	10://Clear old Data on GVL 	
		Lynus_Standards.GVL_Energy.stDataElectricHeatingElements[diNrOfEMS_IN_CP,diNrOfEHE_OUT].bEnabled := FALSE;
			Lynus_Standards.GVL_Energy.stDataElectricHeatingElements[diNrOfEMS_IN_CP,diNrOfEHE_OUT].bIsStepSwitched := FALSE;
				Lynus_Standards.GVL_Energy.stDataElectricHeatingElements[diNrOfEMS_IN_CP,diNrOfEHE_OUT].bIsControllable := FALSE;
					Lynus_Standards.GVL_Energy.stDataElectricHeatingElements[diNrOfEMS_IN_CP,diNrOfEHE_OUT].byPriority := 0;
						Lynus_Standards.GVL_Energy.stDataElectricHeatingElements[diNrOfEMS_IN_CP,diNrOfEHE_OUT].byErrorWarning := 0;
							Lynus_Standards.GVL_Energy.stDataElectricHeatingElements[diNrOfEMS_IN_CP,diNrOfEHE_OUT].byNumberOfSteps := 0;
								Lynus_Standards.GVL_Energy.stDataElectricHeatingElements[diNrOfEMS_IN_CP,diNrOfEHE_OUT].lrPower := 0;
									Lynus_Standards.GVL_Energy.stDataElectricHeatingElements[diNrOfEMS_IN_CP,diNrOfEHE_OUT].lrPowerConsumption := 0;
										Lynus_Standards.GVL_Energy.stDataElectricHeatingElements[diNrOfEMS_IN_CP,diNrOfEHE_OUT].lrPowerProduction := 0;
											FOR byLPGVLSetMaxPower := 1 TO 10 BY 1 DO
												Lynus_Standards.GVL_Energy.stDataElectricHeatingElements[diNrOfEMS_IN_CP,diNrOfEHE_OUT].arrMaxPower[byLPGVLSetMaxPower] := 0;
											END_FOR 
												
		diNrOfEMS_IN_CP := diNrOfEMS_IN;
			//Back to the init step
			iStateGVLData := 0;

END_CASE 	 

IF diNrOfEHE_OUT > 0 AND fbNumberDevice.bNumberIsCalculatet AND diNrOfEMS_IN > 0 THEN
	Lynus_Standards.GVL_Energy.stDataElectricHeatingElements[diNrOfEMS_IN,diNrOfEHE_OUT].bEnabled := fbEHE.stDataEHEOut.bEnabled;
		Lynus_Standards.GVL_Energy.stDataElectricHeatingElements[diNrOfEMS_IN,diNrOfEHE_OUT].bIsStepSwitched := fbEHE.stDataEHEOut.bIsStepSwitched;
			Lynus_Standards.GVL_Energy.stDataElectricHeatingElements[diNrOfEMS_IN,diNrOfEHE_OUT].bIsControllable := TRUE;
				Lynus_Standards.GVL_Energy.stDataElectricHeatingElements[diNrOfEMS_IN,diNrOfEHE_OUT].byPriority := fbEHE.stDataEHEOut.byPriority;
					Lynus_Standards.GVL_Energy.stDataElectricHeatingElements[diNrOfEMS_IN,diNrOfEHE_OUT].byErrorWarning := fbEHE.stDataEHEOut.byErrorWarning;
						Lynus_Standards.GVL_Energy.stDataElectricHeatingElements[diNrOfEMS_IN,diNrOfEHE_OUT].byNumberOfSteps := fbEHE.stDataEHEOut.byNumberOfSteps;
							Lynus_Standards.GVL_Energy.stDataElectricHeatingElements[diNrOfEMS_IN,diNrOfEHE_OUT].lrPower := fbEHE.stDataEHEOut.lrPower;
								Lynus_Standards.GVL_Energy.stDataElectricHeatingElements[diNrOfEMS_IN,diNrOfEHE_OUT].lrPowerConsumption := fbEHE.stDataEHEOut.lrPowerConsumption;
									Lynus_Standards.GVL_Energy.stDataElectricHeatingElements[diNrOfEMS_IN,diNrOfEHE_OUT].lrPowerProduction := fbEHE.stDataEHEOut.lrPowerProduction;
										Lynus_Standards.GVL_Energy.stDataElectricHeatingElements[diNrOfEMS_IN,diNrOfEHE_OUT].arrMaxPower := fbEHE.stDataEHEOut.arrMaxPower;
END_IF			
		
(*----------------------------------------------------------Save persistent data----------------------------------------------------------------*)

arrPD[1](lrValue:= BOOL_TO_LREAL(bEnable), bEventBasedActive=> );
arrPD[2](lrValue:= BOOL_TO_LREAL(bPowerDataInvers), bEventBasedActive=> );
arrPD[3](lrValue:= DINT_TO_LREAL(diNrOfEMS_IN), bEventBasedActive=> );
arrPD[4](lrValue:= DINT_TO_LREAL(diNrOfEM_IN_EHE), bEventBasedActive=> );
arrPD[5](lrValue:= DINT_TO_LREAL(diNrOfTempS_IN), bEventBasedActive=> );
arrPD[6](lrValue:= REAL_TO_LREAL(stSetupEHE.rMaxPower1), bEventBasedActive=> );
arrPD[7](lrValue:= REAL_TO_LREAL(stSetupEHE.rMaxPower2), bEventBasedActive=> );
arrPD[8](lrValue:= REAL_TO_LREAL(stSetupEHE.rMaxPower3), bEventBasedActive=> );
arrPD[9](lrValue:= REAL_TO_LREAL(stSetupEHE.rMaxPower4), bEventBasedActive=> );
arrPD[10](lrValue:= REAL_TO_LREAL(stSetupEHE.rMaxPower5), bEventBasedActive=> );
arrPD[11](lrValue:= REAL_TO_LREAL(stSetupEHE.rMaxPower6), bEventBasedActive=> );
arrPD[12](lrValue:= REAL_TO_LREAL(stSetupEHE.rMaxPower7), bEventBasedActive=> );
arrPD[13](lrValue:= REAL_TO_LREAL(stSetupEHE.rMaxPower8), bEventBasedActive=> );
arrPD[14](lrValue:= REAL_TO_LREAL(stSetupEHE.rMaxPower9), bEventBasedActive=> );
arrPD[15](lrValue:= REAL_TO_LREAL(stSetupEHE.rMaxPower10), bEventBasedActive=> );
arrPD[16](lrValue:= BOOL_TO_LREAL(stSetupEHE.bDisableLegionellaPr), bEventBasedActive=> );
arrPD[17](lrValue:= BOOL_TO_LREAL(stSetupEHE.bManualyOn), bEventBasedActive=> );
arrPD[18](lrValue:= BOOL_TO_LREAL(stSetupEHE.bOnEmergPowerOff), bEventBasedActive=> );
arrPD[19](lrValue:= BOOL_TO_LREAL(stSetupEHE.bTimeEnabled), bEventBasedActive=> );
arrPD[20](lrValue:= BYTE_TO_LREAL(stSetupEHE.byDisableSOC), bEventBasedActive=> );
arrPD[21](lrValue:= BYTE_TO_LREAL(stSetupEHE.byEnableSOC), bEventBasedActive=> );
arrPD[22](lrValue:= BYTE_TO_LREAL(stSetupEHE.byHourOff), bEventBasedActive=> );
arrPD[23](lrValue:= BYTE_TO_LREAL(stSetupEHE.byHourOn), bEventBasedActive=> );
arrPD[24](lrValue:= BYTE_TO_LREAL(stSetupEHE.byManualyTargetPower), bEventBasedActive=> );
arrPD[25](lrValue:= BYTE_TO_LREAL(stSetupEHE.byMinutesOff), bEventBasedActive=> );
arrPD[26](lrValue:= BYTE_TO_LREAL(stSetupEHE.byMinutesOn), bEventBasedActive=> );
arrPD[27](lrValue:= BYTE_TO_LREAL(stSetupEHE.byPriority), bEventBasedActive=> );
arrPD[28](lrValue:= UINT_TO_LREAL(stSetupEHE.uiTargetTempMax), bEventBasedActive=> );
arrPD[29](lrValue:= UINT_TO_LREAL(stSetupEHE.uiTargetTempOff), bEventBasedActive=> );
arrPD[30](lrValue:= UINT_TO_LREAL(stSetupEHE.uiTargetTempOn), bEventBasedActive=> );
arrPD[31](lrValue:= DINT_TO_LREAL(diNrOfEMS_IN_CP), bEventBasedActive=> );
arrPD[32](lrValue:= BOOL_TO_LREAL(bNoLinear), bEventBasedActive=> );
arrPD[33](lrValue:= REAL_TO_LREAL(arrTableOfInterpolationPoints[1]), bEventBasedActive=> );
arrPD[34](lrValue:= REAL_TO_LREAL(arrTableOfInterpolationPoints[2]), bEventBasedActive=> );
arrPD[35](lrValue:= REAL_TO_LREAL(arrTableOfInterpolationPoints[3]), bEventBasedActive=> );
arrPD[36](lrValue:= REAL_TO_LREAL(arrTableOfInterpolationPoints[4]), bEventBasedActive=> );
arrPD[37](lrValue:= REAL_TO_LREAL(arrTableOfInterpolationPoints[5]), bEventBasedActive=> );
arrPD[38](lrValue:= REAL_TO_LREAL(arrTableOfInterpolationPoints[6]), bEventBasedActive=> );
arrPD[39](lrValue:= REAL_TO_LREAL(arrTableOfInterpolationPoints[7]), bEventBasedActive=> );
arrPD[40](lrValue:= REAL_TO_LREAL(arrTableOfInterpolationPoints[8]), bEventBasedActive=> );
arrPD[41](lrValue:= REAL_TO_LREAL(arrTableOfInterpolationPoints[9]), bEventBasedActive=> );
arrPD[42](lrValue:= REAL_TO_LREAL(arrTableOfInterpolationPoints[10]), bEventBasedActive=> );

END_FUNCTION_BLOCK

// ---- FBs/Electric Heating Element/OnOff/FB_EHE_OnOff.TcPOU
FUNCTION_BLOCK FB_EHE_OnOff
VAR_INPUT PERSISTENT
	bEnable									: BOOL;																							//{#lynus.ag#()} //Enable the Fuctionblock and his logic
	bPowerDataInvers						: BOOL;																							//With True its possible to invert all received power data from the electric meter
	diNrOfEMS_IN							: DINT;																							//Number of EMS what control this Device.
	diNrOfEM_IN_EHE							: DINT;																							//Number of the electric meter for incoming power data. (Power Data for this Device)
	diNrOfTempS_IN							: DINT;																							//Number of the Temperature Sensor for incoming temperature data. (Temperature for the Service wather buffer)
	stSetupEHE								: ST_Setup_EHE := (uiTargetTempOn := 35, uiTargetTempOff := 50, uiTargetTempMax := 62);			//{#lynus.ag#()} //Setup electric heating element
END_VAR
VAR_INPUT
END_VAR
VAR_OUTPUT
	stDataEHE								: ST_EHE_Output;																				//{#lynus.ag#()} //Electric heating element output data
	diNrOfEHE_OUT							: DINT;																							//Active Number from the Electric heating element for using on other functions
	rTargetPowerForExtFunc					: REAL;																							//Target Power from 0% to +100% to use on a external Function
END_VAR
VAR
	{attribute 'conditionalshow'}
	fbEHE									: FB_ElectricHeatingElement;																	//Function block for electric heating element
	{attribute 'hide'}
	fbNumberDevice							: FB_NumberOfDevice;																			//Function block to calcualte the number of the Device
	fbDIExternalLock						: FB_XL1XXX_DI;																					//Digital Input from external loock signal
	fbDOOnOffEHE							: FB_XL2XXX_DO;																					//Digital Output to swtich on and off the EHE
	{attribute 'hide'}
	timDissableFunctions					: TON;																							//Timer to dissable the Function after Lynus_Standards.Constants_General.tTimeDissableLynusFunctions Days without connection to the Lynus Cloud
	{attribute 'hide'}
	timResetConnectionOnGVL					: TON;																							//Timer to try reset the connection Flag on the GVL. (When somebody delete the Connection Function and make only a onlinechange)
	{attribute 'hide'}
	timGetTime								: TON;																							//Timer to activate the function tho read out the windows system time
	{attribute 'hide'}
	fbGetSystemTime							: NT_GetTime;																					//Function to read out the windows system time on the local plc
	{attribute 'hide'}
	arrPD									: ARRAY[1..31] OF FB_PersistentData_Number;														//Function to save persistent data 
	{attribute 'hide'}
	byLPTargetPowerTo0						: BYTE;																							//Loop to set the target power from the ems and the max power from the settings for arr[2] to arr[10] to 0 because its only a onOff EHE
	{attribute 'hide'}
	byLPGVLSetMaxPower						: BYTE;																							//Loop to send the max power from the EHE to the GVL
	{attribute 'hide'}
	byWaitInStep							: BYTE;																							//Wait in Step before start to clean data on PLC
	{attribute 'hide'}
	iStateGVLData							: INT;																							//State machine to handle the data on the GVL
	{attribute 'hide'}
	diNumberOfActiveBatterys				: DINT;																							//Number of active batterys
	{attribute 'hide'}
	diNumberOfBatteryInverterInEPO			: DINT;																							//Number of battery inverters that work in Emergency Power operation 
	{attribute 'hide'}
	diCounterForGVL							: DINT;																							//Counter to clean old data on GVL
	{attribute 'hide'}
	diLPForGVL								: DINT;																							//Loop to clean old data on GVL
	{attribute 'hide'}
	dwSumSOC								: DWORD;																						//Sum of the SOC from all batterys
	{attribute 'hide'}
	lrGridPower								: LREAL;																						//Grid power in kW
	{attribute 'hide'}
	lrSizeGridConnection					: LREAL;																						//Size of the complete grid connection
	{attribute 'hide'}
	liLPBatteryData							: LINT;																							//Loop to check some data from batterys
	{attribute 'hide'}
	liLPInEPO								: LINT;																							//Loop to check if 1 or more battery inverters build a island grid
	{attribute 'hide'}
	liLPGridData							: LINT;																							//Loop to check some grid data																				
END_VAR
VAR PERSISTENT
	{attribute 'conditionalshow'}
	diNrOfEMS_IN_CP							: DINT;																							//Number of EMS what control this Device to compare with the original
END_VAR

//Creator : Kai Ebensperger
//Company : Lynus AG
//Date : 19.05.2021
//Version : 1.0.0.0

//With this function block its possible to switch on and off a electric heating element
//The output signal to switch on and off is a digital output signal
//With this function block its not possible to control the EHE with a target power value because we didn't have a active communication to the EHE
//With the Nr from the Electric Meter its possible to send the data fromt the electric meter directly to the EHE function to display it

//NOTE for diNr.....Designation => 
//_IN = Here Data come in from other Functions or go out to other functions about the GVL
//_OUT = Here Data go out to other functions about the GVL

(*------------------------------------------------------------Limits----------------------------------------------------------------------------------*)

diNrOfEMS_IN := LIMIT(0,diNrOfEMS_IN,Constants_Energy.diMaxNumberOfEMS);
	diNrOfEM_IN_EHE := LIMIT(0,diNrOfEM_IN_EHE,Constants_Energy.diMaxNumberOfElectricMeters);
		diNrOfTempS_IN := LIMIT(0,diNrOfTempS_IN,Constants_Sensors.diMaxNumberOfTemperatureSensors);
			
(*------------------------------------------------------------------Power Data----------------------------------------------------------------------------*)

IF NOT bPowerDataInvers THEN
	fbEHE.lrCounterEnergyT1_Consumption := Lynus_Standards.GVL_Energy.stDataElectricMeters[diNrOfEM_IN_EHE].lrCounterEnergyT1_Production * 1000;
	fbEHE.lrCounterEnergyT2_Consumption := Lynus_Standards.GVL_Energy.stDataElectricMeters[diNrOfEM_IN_EHE].lrCounterEnergyT2_Production * 1000;
	fbEHE.lrCounterEnergyT1_Production := Lynus_Standards.GVL_Energy.stDataElectricMeters[diNrOfEM_IN_EHE].lrCounterEnergyT1_Consumption * 1000;
	fbEHE.lrCounterEnergyT2_Production := Lynus_Standards.GVL_Energy.stDataElectricMeters[diNrOfEM_IN_EHE].lrCounterEnergyT1_Consumption * 1000;
	fbEHE.lrTotalCounterEnergy_Consumption := Lynus_Standards.GVL_Energy.stDataElectricMeters[diNrOfEM_IN_EHE].lrTotalCounterEnergy_Production * 1000;
	fbEHE.lrTotalCounterEnergy_Production := Lynus_Standards.GVL_Energy.stDataElectricMeters[diNrOfEM_IN_EHE].lrTotalCounterEnergy_Consumption * 1000;
		fbEHE.lrPowerEHE := (Lynus_Standards.GVL_Energy.stDataElectricMeters[diNrOfEM_IN_EHE].lrPower * 1000) * - 1;
ELSE
	fbEHE.lrCounterEnergyT1_Consumption := Lynus_Standards.GVL_Energy.stDataElectricMeters[diNrOfEM_IN_EHE].lrCounterEnergyT1_Consumption * 1000;
	fbEHE.lrCounterEnergyT2_Consumption := Lynus_Standards.GVL_Energy.stDataElectricMeters[diNrOfEM_IN_EHE].lrCounterEnergyT2_Consumption * 1000;
	fbEHE.lrCounterEnergyT1_Production := Lynus_Standards.GVL_Energy.stDataElectricMeters[diNrOfEM_IN_EHE].lrCounterEnergyT1_Production * 1000;
	fbEHE.lrCounterEnergyT2_Production := Lynus_Standards.GVL_Energy.stDataElectricMeters[diNrOfEM_IN_EHE].lrCounterEnergyT2_Production * 1000;
	fbEHE.lrTotalCounterEnergy_Consumption := Lynus_Standards.GVL_Energy.stDataElectricMeters[diNrOfEM_IN_EHE].lrTotalCounterEnergy_Consumption * 1000;
	fbEHE.lrTotalCounterEnergy_Production := Lynus_Standards.GVL_Energy.stDataElectricMeters[diNrOfEM_IN_EHE].lrTotalCounterEnergy_Production * 1000;
		fbEHE.lrPowerEHE := Lynus_Standards.GVL_Energy.stDataElectricMeters[diNrOfEM_IN_EHE].lrPower * 1000;
END_IF

(*-------------------------------------------------------------Calcualte the number of EHE---------------------------------------------------------------*)

fbNumberDevice(
	diActualNumberOfDevices:= Lynus_Standards.GVL_Energy.stNumberOfDevices.diNumberOfEHE, 
	diMaxNumberOfDevices:= Constants_Energy.diMaxNumberOfElectricHeatingElements, 
	udiCounterOnlineChange:= TwinCAT_SystemInfoVarList._AppInfo.OnlineChangeCnt, 
	bNumberIsCalculatet=> , 
	bFPNumberIsCalculatet=> , 
	bOnlineChange=> , 
	diNumberForThisDevice=> diNrOfEHE_OUT, 
	diNumberOfTotalDevices=> );

//Write new Numer on GVL
IF fbNumberDevice.bFPNumberIsCalculatet THEN
	Lynus_Standards.GVL_Energy.stNumberOfDevices.diNumberOfEHE := fbNumberDevice.diNumberOfTotalDevices;	
END_IF 

//Delete old Number on GVL
IF fbNumberDevice.bOnlineChange THEN 
	Lynus_Standards.GVL_Energy.stNumberOfDevices.diNumberOfEHE := diNrOfEHE_OUT;	
		iStateGVLData := 1; 
END_IF

(*-------------------------------------------------------------Get the local windows system time for this plc---------------------------------------------------------------*)
timGetTime(IN:= bEnable AND NOT timGetTime.Q, PT:= T#30S, Q=> , ET=> );

fbGetSystemTime(
	NETID:= , 
	START:= timGetTime.Q AND NOT fbGetSystemTime.BUSY, 
	TMOUT:= , 
	BUSY=> , 
	ERR=> , 
	ERRID=> , 
	TIMESTR=> );	

fbEHE.stSystemTime.wHour := fbGetSystemTime.TIMESTR.wHour;
	fbEHE.stSystemTime.wMinute := fbGetSystemTime.TIMESTR.wMinute;

(*-------------------------------------------------------------Service from Backend is ready and check the connection to backen for dissabel/enable Function---------------------------------------------------------------*)

//Try to reset the variable for connection on the GVL. When all is normal then the Lynus Mqtt connection function set this variable to true in the next cycle
//When we have no connection to the backend then after Lynus_Standards.Constants_General.tTimeDissableLynusFunctions days the Function is dissabled with all of his functionalities
timResetConnectionOnGVL(IN:= NOT timResetConnectionOnGVL.Q, PT:= T#1H, Q=> , ET=> );
	IF timResetConnectionOnGVL.Q THEN Lynus_Standards.GVL_Communicator.bStateConnectionToEnableFunctions := FALSE; END_IF
		IF NOT Lynus_Standards.GVL_Communicator.bStateConnectionToEnableFunctions THEN timDissableFunctions.IN := TRUE; ELSE timDissableFunctions.IN := FALSE; END_IF  
			timDissableFunctions(IN:= , PT:= Lynus_Standards.Constants_General.tTimeDissableLynusFunctions, Q=> , ET=> );
	
(*------------------------------------------------------------------Error----------------------------------------------------------------------------*)	

IF timDissableFunctions.Q THEN fbEHE.bWarning := TRUE; fbEHE.iWarningCode := 0; ELSE fbEHE.bWarning := FALSE; END_IF 
	IF (Lynus_Standards.GVL_Energy.stNumberOfDevices.diNumberOfEHE > Constants_Energy.diMaxNumberOfElectricHeatingElements) OR 
		(Lynus_Standards.GVL_Sensors.stDataTemperatureSensors[diNrOfTempS_IN].bEnabled AND Lynus_Standards.GVL_Sensors.stDataTemperatureSensors[diNrOfTempS_IN].byErrorWarning = 2) OR
			fbGetSystemTime.ERR THEN 
				fbEHE.bError := TRUE; 
	ELSE 
				fbEHE.bError := FALSE; 
	END_IF

IF Lynus_Standards.GVL_Energy.stNumberOfDevices.diNumberOfEHE > Constants_Energy.diMaxNumberOfElectricHeatingElements THEN fbEHE.iErrorCode := 1;
ELSIF fbGetSystemTime.ERR THEN fbEHE.iErrorCode := 3;
ELSIF Lynus_Standards.GVL_Sensors.stDataTemperatureSensors[diNrOfTempS_IN].bEnabled AND Lynus_Standards.GVL_Sensors.stDataTemperatureSensors[diNrOfTempS_IN].byErrorWarning = 2 THEN fbEHE.iErrorCode := 2;
END_IF

(*------------------------------------------------------------------Logic----------------------------------------------------------------------------*)
	
//Calcualte the total SOC if we have more then 1 battery in our system
diNumberOfActiveBatterys := 0;
	dwSumSOC := 0;
		FOR liLPBatteryData := 1 TO Constants_Energy.diMaxNumberOfBatterys BY 1 DO
			IF Lynus_Standards.GVL_Energy.stDataOfBatterys[diNrOfEMS_IN,liLPBatteryData].bEnabled THEN diNumberOfActiveBatterys := diNumberOfActiveBatterys + 1; END_IF
				dwSumSOC := dwSumSOC + Lynus_Standards.GVL_Energy.stDataOfBatterys[diNrOfEMS_IN,liLPBatteryData].dwSOC;
		END_FOR
	
IF diNumberOfActiveBatterys > 0 THEN
	fbEHE.dwBatterySOC := DINT_TO_DWORD(DWORD_TO_DINT(dwSumSOC) / diNumberOfActiveBatterys);
ELSE
	fbEHE.dwBatterySOC := 100;	//When we have no battery in the ems system
END_IF

//Check if one or more Batterysystems or batteryinverter make island mode
diNumberOfBatteryInverterInEPO := 0;
	FOR liLPInEPO := 1 TO Constants_Energy.diMaxNumberOfBatteryInverters BY 1 DO
		IF Lynus_Standards.GVL_Energy.stDataOfBatteryInverters[diNrOfEMS_IN,liLPInEPO].bWorkOnIslandMode THEN fbEHE.bEPOIsActive := TRUE; diNumberOfBatteryInverterInEPO := diNumberOfBatteryInverterInEPO + 1; END_IF
	END_FOR 
		IF diNumberOfBatteryInverterInEPO <= 0 THEN fbEHE.bEPOIsActive := FALSE; END_IF

//Check the max. power of the grid connection and the sum of grid power
lrSizeGridConnection := 0;
	lrGridPower := 0;
		FOR liLPGridData := 1 TO Constants_Energy.diMaxNumberOfGridConnections BY 1 DO
			lrSizeGridConnection := lrSizeGridConnection + Lynus_Standards.GVL_Energy.stDataGridConnections[diNrOfEMS_IN,liLPGridData].rSizeGridConn;
				lrGridPower := lrGridPower + Lynus_Standards.GVL_Energy.stDataGridConnections[diNrOfEMS_IN,liLPGridData].lrPower;
		END_FOR			
		
//Set the target power from the EMS to the EHE Function
fbEHE.arrTargetPower[1] := Lynus_Standards.GVL_Energy.stDataElectricHeatingElements[diNrOfEMS_IN,diNrOfEHE_OUT].arrTargetPowerEMS[1];

FOR byLPTargetPowerTo0 := 2 TO 10 BY 1 DO
	fbEHE.arrTargetPower[byLPTargetPowerTo0] := 0;
END_FOR
	stSetupEHE.rMaxPower2 := 0;
		stSetupEHE.rMaxPower3 := 0;
			stSetupEHE.rMaxPower4 := 0;
				stSetupEHE.rMaxPower5 := 0;
					stSetupEHE.rMaxPower6 := 0;
						stSetupEHE.rMaxPower7 := 0;
							stSetupEHE.rMaxPower8 := 0;
								stSetupEHE.rMaxPower9 := 0;
									stSetupEHE.rMaxPower10 := 0;

//Digital input for external lock signal
fbDIExternalLock(bInvers:= FALSE, bSignal=> );

//Functionblock EHE
fbEHE.stSetupEHE.bManualyOn := stSetupEHE.bManualyOn;
	IF fbEHE.stSetupEHE.bManualyOn THEN fbEHE.stSetupEHE.byManualyTargetPower := 100; ELSE fbEHE.stSetupEHE.byManualyTargetPower := 0; END_IF
		fbEHE.stSetupEHE.bOnEmergPowerOff := stSetupEHE.bOnEmergPowerOff;
			fbEHE.stSetupEHE.bTimeEnabled := stSetupEHE.bTimeEnabled;
				fbEHE.stSetupEHE.bDisableLegionellaPr := stSetupEHE.bDisableLegionellaPr;	
					fbEHE.stSetupEHE.byPriority := stSetupEHE.byPriority;
						fbEHE.stSetupEHE.byEnableSOC := stSetupEHE.byEnableSOC;
							fbEHE.stSetupEHE.byDisableSOC := stSetupEHE.byDisableSOC;
								fbEHE.stSetupEHE.byHourOn := stSetupEHE.byHourOn;
									fbEHE.stSetupEHE.byMinutesOn := stSetupEHE.byMinutesOn;
										fbEHE.stSetupEHE.byHourOff := stSetupEHE.byHourOff;
											fbEHE.stSetupEHE.byMinutesOff := stSetupEHE.byMinutesOff;
												fbEHE.stSetupEHE.uiTargetTempOn := stSetupEHE.uiTargetTempOn;
													fbEHE.stSetupEHE.uiTargetTempOff := stSetupEHE.uiTargetTempOff;
														fbEHE.stSetupEHE.uiTargetTempMax := stSetupEHE.uiTargetTempMax;
															fbEHE.stSetupEHE.rMaxPower1 := stSetupEHE.rMaxPower1;
																fbEHE.stSetupEHE.rMaxPower2 := stSetupEHE.rMaxPower2;
																	fbEHE.stSetupEHE.rMaxPower3 := stSetupEHE.rMaxPower3;
																		fbEHE.stSetupEHE.rMaxPower4 := stSetupEHE.rMaxPower4;
																			fbEHE.stSetupEHE.rMaxPower5 := stSetupEHE.rMaxPower5;
																				fbEHE.stSetupEHE.rMaxPower6 := stSetupEHE.rMaxPower6;
																					fbEHE.stSetupEHE.rMaxPower7 := stSetupEHE.rMaxPower7;
																						fbEHE.stSetupEHE.rMaxPower8 := stSetupEHE.rMaxPower8;
																							fbEHE.stSetupEHE.rMaxPower9 := stSetupEHE.rMaxPower9;
																								fbEHE.stSetupEHE.rMaxPower10 := stSetupEHE.rMaxPower10;

fbEHE(
	bEnable:= bEnable AND NOT timDissableFunctions.Q,
	bError:= , 
	bIsStepSwitched:= FALSE, 
	bEPOIsActive:= , 
	bExternalLock:= fbDIExternalLock.bSignal, 
	bWriteWithDelay:= TRUE,
	bTimeDissableFunctions:= timDissableFunctions.Q, 
	iErrorCode:= , 
	iWarningCode:= ,
	diNumberOfEHE:= diNrOfEHE_OUT,
	dwBatterySOC:= ,
	lrSizeGridConnection:= lrSizeGridConnection,
	lrGridPower:= lrGridPower, 
	lrTotalCounterEnergy_Consumption:= , 
	lrTotalCounterEnergy_Production:= , 
	lrCounterEnergyT1_Consumption:= , 
	lrCounterEnergyT2_Consumption:= , 
	lrCounterEnergyT1_Production:= , 
	lrCounterEnergyT2_Production:= , 
	lrPowerEHE:= , 
	arrTargetPower:= , 
	rTemperatureInBoiler:= Lynus_Standards.GVL_Sensors.stDataTemperatureSensors[diNrOfTempS_IN].rTemperature, 
	tTimDelayOutput:= T#5S, 
	stSystemTime:= , 
	stSetupEHE:= , 
	stDataEHEOut=> , 
	stDataEHEOutDelay=> stDataEHE);

//Target Power, to use this on a external Function
rTargetPowerForExtFunc := fbEHE.stDataEHEOut.rTargetPower;
	
(*-------------------------------------------------------------------------Output----------------------------------------------------------------------*)

fbDOOnOffEHE(bInvers:= FALSE, bSignal:= fbEHE.stDataEHEOut.bOutputOnOff);

(*-----------------------------------------------------------Handle data to Global structure for the electric heating element-----------------------------------------------------------------*)

//Delte al old Data on GVL after a online change or change on the variable diNrOfEMS_IDOD
IF diNrOfEMS_IN <> diNrOfEMS_IN_CP AND iStateGVLData = 0 THEN iStateGVLData := 10; END_IF 

CASE iStateGVLData OF
	
	0://Init Step
		byWaitInStep := 0;
			diCounterForGVL := 1;
	
	1://Wait for 4 Steps before clean al Data on GVL
		byWaitInStep := byWaitInStep + 1;
			IF byWaitInStep >= 4 AND fbNumberDevice.bNumberIsCalculatet THEN iStateGVLData := 2; END_IF
				//To much Devices, back to the Init step
				IF byWaitInStep >= 4 AND NOT fbNumberDevice.bNumberIsCalculatet THEN iStateGVLData := 0; END_IF	
			
	2://Clear all Data in GVL
		FOR diLPForGVL := 1 TO Constants_Energy.diMaxNumberOfEMS BY 1 DO 
			Lynus_Standards.GVL_Energy.stDataElectricHeatingElements[diLPForGVL,diCounterForGVL].bEnabled := FALSE;
				Lynus_Standards.GVL_Energy.stDataElectricHeatingElements[diLPForGVL,diCounterForGVL].bIsStepSwitched := FALSE;
					Lynus_Standards.GVL_Energy.stDataElectricHeatingElements[diLPForGVL,diCounterForGVL].bIsControllable := FALSE;
						Lynus_Standards.GVL_Energy.stDataElectricHeatingElements[diLPForGVL,diCounterForGVL].byPriority := 0;
							Lynus_Standards.GVL_Energy.stDataElectricHeatingElements[diLPForGVL,diCounterForGVL].byErrorWarning := 0;
								Lynus_Standards.GVL_Energy.stDataElectricHeatingElements[diLPForGVL,diCounterForGVL].byNumberOfSteps := 0;
									Lynus_Standards.GVL_Energy.stDataElectricHeatingElements[diLPForGVL,diCounterForGVL].lrPower := 0;
										Lynus_Standards.GVL_Energy.stDataElectricHeatingElements[diLPForGVL,diCounterForGVL].lrPowerConsumption := 0;
											Lynus_Standards.GVL_Energy.stDataElectricHeatingElements[diLPForGVL,diCounterForGVL].lrPowerProduction := 0;
												FOR byLPGVLSetMaxPower := 1 TO 10 BY 1 DO
													Lynus_Standards.GVL_Energy.stDataElectricHeatingElements[diLPForGVL,diCounterForGVL].arrMaxPower[byLPGVLSetMaxPower] := 0;
												END_FOR 
													//Set also the target value from ems back here to 0 and not in EMS function because EMS is in Standy when we have a online change (Problem when we delete a ems function and make a online change)
													FOR byLPGVLSetMaxPower := 1 TO 10 BY 1 DO
														Lynus_Standards.GVL_Energy.stDataElectricHeatingElements[diLPForGVL,diCounterForGVL].arrTargetPowerEMS[byLPGVLSetMaxPower] := 0;	
													END_FOR
		END_FOR
			diCounterForGVL := diCounterForGVL + 1;
				diCounterForGVL := LIMIT(0,diCounterForGVL,Constants_Energy.diMaxNumberOfElectricHeatingElements);
					//Back to the init step
					IF diCounterForGVL >= Constants_Energy.diMaxNumberOfElectricHeatingElements THEN iStateGVLData := 0; END_IF

	10://Clear old Data on GVL 	
		Lynus_Standards.GVL_Energy.stDataElectricHeatingElements[diNrOfEMS_IN_CP,diNrOfEHE_OUT].bEnabled := FALSE;
			Lynus_Standards.GVL_Energy.stDataElectricHeatingElements[diNrOfEMS_IN_CP,diNrOfEHE_OUT].bIsStepSwitched := FALSE;
				Lynus_Standards.GVL_Energy.stDataElectricHeatingElements[diNrOfEMS_IN_CP,diNrOfEHE_OUT].bIsControllable := FALSE;
					Lynus_Standards.GVL_Energy.stDataElectricHeatingElements[diNrOfEMS_IN_CP,diNrOfEHE_OUT].byPriority := 0;
						Lynus_Standards.GVL_Energy.stDataElectricHeatingElements[diNrOfEMS_IN_CP,diNrOfEHE_OUT].byErrorWarning := 0;
							Lynus_Standards.GVL_Energy.stDataElectricHeatingElements[diNrOfEMS_IN_CP,diNrOfEHE_OUT].byNumberOfSteps := 0;
								Lynus_Standards.GVL_Energy.stDataElectricHeatingElements[diNrOfEMS_IN_CP,diNrOfEHE_OUT].lrPower := 0;
									Lynus_Standards.GVL_Energy.stDataElectricHeatingElements[diNrOfEMS_IN_CP,diNrOfEHE_OUT].lrPowerConsumption := 0;
										Lynus_Standards.GVL_Energy.stDataElectricHeatingElements[diNrOfEMS_IN_CP,diNrOfEHE_OUT].lrPowerProduction := 0;
											FOR byLPGVLSetMaxPower := 1 TO 10 BY 1 DO
												Lynus_Standards.GVL_Energy.stDataElectricHeatingElements[diNrOfEMS_IN_CP,diNrOfEHE_OUT].arrMaxPower[byLPGVLSetMaxPower] := 0;
											END_FOR 
												
		diNrOfEMS_IN_CP := diNrOfEMS_IN;
			//Back to the init step
			iStateGVLData := 0;

END_CASE 	 

IF diNrOfEHE_OUT > 0 AND fbNumberDevice.bNumberIsCalculatet AND diNrOfEMS_IN > 0 THEN
	Lynus_Standards.GVL_Energy.stDataElectricHeatingElements[diNrOfEMS_IN,diNrOfEHE_OUT].bEnabled := fbEHE.stDataEHEOut.bEnabled;
		Lynus_Standards.GVL_Energy.stDataElectricHeatingElements[diNrOfEMS_IN,diNrOfEHE_OUT].bIsStepSwitched := fbEHE.stDataEHEOut.bIsStepSwitched;
			Lynus_Standards.GVL_Energy.stDataElectricHeatingElements[diNrOfEMS_IN,diNrOfEHE_OUT].bIsControllable := FALSE;
				Lynus_Standards.GVL_Energy.stDataElectricHeatingElements[diNrOfEMS_IN,diNrOfEHE_OUT].byPriority := fbEHE.stDataEHEOut.byPriority;
					Lynus_Standards.GVL_Energy.stDataElectricHeatingElements[diNrOfEMS_IN,diNrOfEHE_OUT].byErrorWarning := fbEHE.stDataEHEOut.byErrorWarning;
						Lynus_Standards.GVL_Energy.stDataElectricHeatingElements[diNrOfEMS_IN,diNrOfEHE_OUT].byNumberOfSteps := fbEHE.stDataEHEOut.byNumberOfSteps;
							Lynus_Standards.GVL_Energy.stDataElectricHeatingElements[diNrOfEMS_IN,diNrOfEHE_OUT].lrPower := fbEHE.stDataEHEOut.lrPower;
								Lynus_Standards.GVL_Energy.stDataElectricHeatingElements[diNrOfEMS_IN,diNrOfEHE_OUT].lrPowerConsumption := fbEHE.stDataEHEOut.lrPowerConsumption;
									Lynus_Standards.GVL_Energy.stDataElectricHeatingElements[diNrOfEMS_IN,diNrOfEHE_OUT].lrPowerProduction := fbEHE.stDataEHEOut.lrPowerProduction;
										Lynus_Standards.GVL_Energy.stDataElectricHeatingElements[diNrOfEMS_IN,diNrOfEHE_OUT].arrMaxPower := fbEHE.stDataEHEOut.arrMaxPower;
END_IF			

(*----------------------------------------------------------Save persistent data----------------------------------------------------------------*)

arrPD[1](lrValue:= BOOL_TO_LREAL(bEnable), bEventBasedActive=> );
arrPD[2](lrValue:= BOOL_TO_LREAL(bPowerDataInvers), bEventBasedActive=> );
arrPD[3](lrValue:= DINT_TO_LREAL(diNrOfEMS_IN), bEventBasedActive=> );
arrPD[4](lrValue:= DINT_TO_LREAL(diNrOfEM_IN_EHE), bEventBasedActive=> );
arrPD[5](lrValue:= DINT_TO_LREAL(diNrOfTempS_IN), bEventBasedActive=> );
arrPD[6](lrValue:= REAL_TO_LREAL(stSetupEHE.rMaxPower1), bEventBasedActive=> );
arrPD[7](lrValue:= REAL_TO_LREAL(stSetupEHE.rMaxPower2), bEventBasedActive=> );
arrPD[8](lrValue:= REAL_TO_LREAL(stSetupEHE.rMaxPower3), bEventBasedActive=> );
arrPD[9](lrValue:= REAL_TO_LREAL(stSetupEHE.rMaxPower4), bEventBasedActive=> );
arrPD[10](lrValue:= REAL_TO_LREAL(stSetupEHE.rMaxPower5), bEventBasedActive=> );
arrPD[11](lrValue:= REAL_TO_LREAL(stSetupEHE.rMaxPower6), bEventBasedActive=> );
arrPD[12](lrValue:= REAL_TO_LREAL(stSetupEHE.rMaxPower7), bEventBasedActive=> );
arrPD[13](lrValue:= REAL_TO_LREAL(stSetupEHE.rMaxPower8), bEventBasedActive=> );
arrPD[14](lrValue:= REAL_TO_LREAL(stSetupEHE.rMaxPower9), bEventBasedActive=> );
arrPD[15](lrValue:= REAL_TO_LREAL(stSetupEHE.rMaxPower10), bEventBasedActive=> );
arrPD[16](lrValue:= BOOL_TO_LREAL(stSetupEHE.bDisableLegionellaPr), bEventBasedActive=> );
arrPD[17](lrValue:= BOOL_TO_LREAL(stSetupEHE.bManualyOn), bEventBasedActive=> );
arrPD[18](lrValue:= BOOL_TO_LREAL(stSetupEHE.bOnEmergPowerOff), bEventBasedActive=> );
arrPD[19](lrValue:= BOOL_TO_LREAL(stSetupEHE.bTimeEnabled), bEventBasedActive=> );
arrPD[20](lrValue:= BYTE_TO_LREAL(stSetupEHE.byDisableSOC), bEventBasedActive=> );
arrPD[21](lrValue:= BYTE_TO_LREAL(stSetupEHE.byEnableSOC), bEventBasedActive=> );
arrPD[22](lrValue:= BYTE_TO_LREAL(stSetupEHE.byHourOff), bEventBasedActive=> );
arrPD[23](lrValue:= BYTE_TO_LREAL(stSetupEHE.byHourOn), bEventBasedActive=> );
arrPD[24](lrValue:= BYTE_TO_LREAL(stSetupEHE.byManualyTargetPower), bEventBasedActive=> );
arrPD[25](lrValue:= BYTE_TO_LREAL(stSetupEHE.byMinutesOff), bEventBasedActive=> );
arrPD[26](lrValue:= BYTE_TO_LREAL(stSetupEHE.byMinutesOn), bEventBasedActive=> );
arrPD[27](lrValue:= BYTE_TO_LREAL(stSetupEHE.byPriority), bEventBasedActive=> );
arrPD[28](lrValue:= UINT_TO_LREAL(stSetupEHE.uiTargetTempMax), bEventBasedActive=> );
arrPD[29](lrValue:= UINT_TO_LREAL(stSetupEHE.uiTargetTempOff), bEventBasedActive=> );
arrPD[30](lrValue:= UINT_TO_LREAL(stSetupEHE.uiTargetTempOn), bEventBasedActive=> );
arrPD[31](lrValue:= DINT_TO_LREAL(diNrOfEMS_IN_CP), bEventBasedActive=> );

END_FUNCTION_BLOCK

// ---- FBs/Electric Heating Element/Step Switched AO/FB_EHE_StepSwitched_AO.TcPOU
FUNCTION_BLOCK FB_EHE_StepSwitched_AO
VAR_INPUT PERSISTENT
	bEnable									: BOOL;																							//{#lynus.ag#()} //Enable the Fuctionblock and his logic
	bPowerDataInvers						: BOOL;																							//With True its possible to invert all received power data from the electric meter
	diNrOfEMS_IN							: DINT;																							//Number of EMS what control this Device.
	diNrOfEM_IN_EHE							: DINT;																							//Number of the electric meter for incoming power data. (Power Data for this Device)
	diNrOfTempS_IN							: DINT;																							//Number of the Temperature Sensor for incoming temperature data. (Temperature for the Service wather buffer)
	stSetupEHE								: ST_Setup_EHE := (uiTargetTempOn := 35, uiTargetTempOff := 50, uiTargetTempMax := 62);			//{#lynus.ag#()} //Setup electric heating element
END_VAR
VAR_INPUT
END_VAR
VAR_OUTPUT
	stDataEHE								: ST_EHE_Output;																				//{#lynus.ag#()} //Electric heating element output data
	diNrOfEHE_OUT							: DINT;																							//Active Number from the Electric heating element for using on other functions
	rTargetPowerForExtFunc					: REAL;																							//Target Power from 0% to +100% to use on a external Function
END_VAR
VAR
	{attribute 'conditionalshow'}
	fbEHE									: FB_ElectricHeatingElement;																	//Function block for electric heating element
	{attribute 'hide'}
	fbNumberDevice							: FB_NumberOfDevice;																			//Function block to calcualte the number of the Device
	fbDIExternalLock						: FB_XL1XXX_DI;																					//Digital Input from external loock signal
	fbAOEHE									: FB_XL4XXX_AO;																					//Analog Output to swtich on and off and controll the EHE
	{attribute 'hide'}
	timDissableFunctions					: TON;																							//Timer to dissable the Function after Lynus_Standards.Constants_General.tTimeDissableLynusFunctions Days without connection to the Lynus Cloud
	{attribute 'hide'}
	timResetConnectionOnGVL					: TON;																							//Timer to try reset the connection Flag on the GVL. (When somebody delete the Connection Function and make only a onlinechange)
	{attribute 'hide'}
	timGetTime								: TON;																							//Timer to activate the function tho read out the windows system time
	{attribute 'hide'}
	fbGetSystemTime							: NT_GetTime;																					//Function to read out the windows system time on the local plc
	{attribute 'hide'}
	arrPD									: ARRAY[1..31] OF FB_PersistentData_Number;														//Function to save persistent data 
	{attribute 'hide'}
	byLPGVLSetMaxPower						: BYTE;																							//Loop to send the max power from the EHE to the GVL
	{attribute 'hide'}
	byWaitInStep							: BYTE;																							//Wait in Step before start to clean data on PLC
	{attribute 'hide'}
	iStateGVLData							: INT;																							//State machine to handle the data on the GVL
	{attribute 'hide'}
	diNumberOfActiveBatterys				: DINT;																							//Number of active batterys
	{attribute 'hide'}
	diNumberOfBatteryInverterInEPO			: DINT;																							//Number of battery inverters that work in Emergency Power operation 
	{attribute 'hide'}
	diCounterForGVL							: DINT;																							//Counter to clean old data on GVL
	{attribute 'hide'}
	diLPForGVL								: DINT;																							//Loop to clean old data on GVL
	{attribute 'hide'}
	dwSumSOC								: DWORD;																						//Sum of the SOC from all batterys
	{attribute 'hide'}
	lrGridPower								: LREAL;																						//Grid power in kW
	{attribute 'hide'}
	lrSizeGridConnection					: LREAL;																						//Size of the complete grid connection
	{attribute 'hide'}
	liLPBatteryData							: LINT;																							//Loop to check some data from batterys
	{attribute 'hide'}
	liLPInEPO								: LINT;																							//Loop to check if 1 or more battery inverters build a island grid
	{attribute 'hide'}
	liLPGridData							: LINT;																							//Loop to check some grid data																				
END_VAR
VAR PERSISTENT
	{attribute 'conditionalshow'}
	diNrOfEMS_IN_CP							: DINT;																							//Number of EMS what control this Device to compare with the original
END_VAR

//Creator : Kai Ebensperger
//Company : Lynus AG
//Date : 19.05.2021
//Version : 1.0.0.0

//With this function block its possible to switch on and off a electric heating element
//The output signal to switch on and off is a analog output signal. (0-10V or 4-20mA)
//With this function block its possible to control the EHE with a target power value over the analog signal. The output signal is step switched. (So for example 10% target power is step 1 wit 1kW, 20% is step 2 with 1kW and so on....)
//With the Nr from the Electric Meter its possible to send the data fromt the electric meter directly to the EHE function to display it

//NOTE for diNr.....Designation => 
//_IN = Here Data come in from other Functions or go out to other functions about the GVL
//_OUT = Here Data go out to other functions about the GVL


(*------------------------------------------------------------Limits----------------------------------------------------------------------------------*)

diNrOfEMS_IN := LIMIT(0,diNrOfEMS_IN,Constants_Energy.diMaxNumberOfEMS);
	diNrOfEM_IN_EHE := LIMIT(0,diNrOfEM_IN_EHE,Constants_Energy.diMaxNumberOfElectricMeters);
		diNrOfTempS_IN := LIMIT(0,diNrOfTempS_IN,Constants_Sensors.diMaxNumberOfTemperatureSensors);
			
(*------------------------------------------------------------------Power Data----------------------------------------------------------------------------*)

IF NOT bPowerDataInvers THEN
	fbEHE.lrCounterEnergyT1_Consumption := Lynus_Standards.GVL_Energy.stDataElectricMeters[diNrOfEM_IN_EHE].lrCounterEnergyT1_Production * 1000;
	fbEHE.lrCounterEnergyT2_Consumption := Lynus_Standards.GVL_Energy.stDataElectricMeters[diNrOfEM_IN_EHE].lrCounterEnergyT2_Production * 1000;
	fbEHE.lrCounterEnergyT1_Production := Lynus_Standards.GVL_Energy.stDataElectricMeters[diNrOfEM_IN_EHE].lrCounterEnergyT1_Consumption * 1000;
	fbEHE.lrCounterEnergyT2_Production := Lynus_Standards.GVL_Energy.stDataElectricMeters[diNrOfEM_IN_EHE].lrCounterEnergyT1_Consumption * 1000;
	fbEHE.lrTotalCounterEnergy_Consumption := Lynus_Standards.GVL_Energy.stDataElectricMeters[diNrOfEM_IN_EHE].lrTotalCounterEnergy_Production * 1000;
	fbEHE.lrTotalCounterEnergy_Production := Lynus_Standards.GVL_Energy.stDataElectricMeters[diNrOfEM_IN_EHE].lrTotalCounterEnergy_Consumption * 1000;
		fbEHE.lrPowerEHE := (Lynus_Standards.GVL_Energy.stDataElectricMeters[diNrOfEM_IN_EHE].lrPower * 1000) * - 1;
ELSE
	fbEHE.lrCounterEnergyT1_Consumption := Lynus_Standards.GVL_Energy.stDataElectricMeters[diNrOfEM_IN_EHE].lrCounterEnergyT1_Consumption * 1000;
	fbEHE.lrCounterEnergyT2_Consumption := Lynus_Standards.GVL_Energy.stDataElectricMeters[diNrOfEM_IN_EHE].lrCounterEnergyT2_Consumption * 1000;
	fbEHE.lrCounterEnergyT1_Production := Lynus_Standards.GVL_Energy.stDataElectricMeters[diNrOfEM_IN_EHE].lrCounterEnergyT1_Production * 1000;
	fbEHE.lrCounterEnergyT2_Production := Lynus_Standards.GVL_Energy.stDataElectricMeters[diNrOfEM_IN_EHE].lrCounterEnergyT2_Production * 1000;
	fbEHE.lrTotalCounterEnergy_Consumption := Lynus_Standards.GVL_Energy.stDataElectricMeters[diNrOfEM_IN_EHE].lrTotalCounterEnergy_Consumption * 1000;
	fbEHE.lrTotalCounterEnergy_Production := Lynus_Standards.GVL_Energy.stDataElectricMeters[diNrOfEM_IN_EHE].lrTotalCounterEnergy_Production * 1000;
		fbEHE.lrPowerEHE := Lynus_Standards.GVL_Energy.stDataElectricMeters[diNrOfEM_IN_EHE].lrPower * 1000;
END_IF

(*-------------------------------------------------------------Calcualte the number of EHE---------------------------------------------------------------*)

fbNumberDevice(
	diActualNumberOfDevices:= Lynus_Standards.GVL_Energy.stNumberOfDevices.diNumberOfEHE, 
	diMaxNumberOfDevices:= Constants_Energy.diMaxNumberOfElectricHeatingElements, 
	udiCounterOnlineChange:= TwinCAT_SystemInfoVarList._AppInfo.OnlineChangeCnt, 
	bNumberIsCalculatet=> , 
	bFPNumberIsCalculatet=> , 
	bOnlineChange=> , 
	diNumberForThisDevice=> diNrOfEHE_OUT, 
	diNumberOfTotalDevices=> );

//Write new Numer on GVL
IF fbNumberDevice.bFPNumberIsCalculatet THEN
	Lynus_Standards.GVL_Energy.stNumberOfDevices.diNumberOfEHE := fbNumberDevice.diNumberOfTotalDevices;	
END_IF 

//Delete old Number on GVL
IF fbNumberDevice.bOnlineChange THEN 
	Lynus_Standards.GVL_Energy.stNumberOfDevices.diNumberOfEHE := diNrOfEHE_OUT;	
		iStateGVLData := 1; 
END_IF

(*-------------------------------------------------------------Get the local windows system time for this plc---------------------------------------------------------------*)
timGetTime(IN:= bEnable AND NOT timGetTime.Q, PT:= T#30S, Q=> , ET=> );

fbGetSystemTime(
	NETID:= , 
	START:= timGetTime.Q AND NOT fbGetSystemTime.BUSY, 
	TMOUT:= , 
	BUSY=> , 
	ERR=> , 
	ERRID=> , 
	TIMESTR=> );	

fbEHE.stSystemTime.wHour := fbGetSystemTime.TIMESTR.wHour;
	fbEHE.stSystemTime.wMinute := fbGetSystemTime.TIMESTR.wMinute;

(*-------------------------------------------------------------Service from Backend is ready and check the connection to backen for dissabel/enable Function---------------------------------------------------------------*)

//Try to reset the variable for connection on the GVL. When all is normal then the Lynus Mqtt connection function set this variable to true in the next cycle
//When we have no connection to the backend then after Lynus_Standards.Constants_General.tTimeDissableLynusFunctions days the Function is dissabled with all of his functionalities
timResetConnectionOnGVL(IN:= NOT timResetConnectionOnGVL.Q, PT:= T#1H, Q=> , ET=> );
	IF timResetConnectionOnGVL.Q THEN Lynus_Standards.GVL_Communicator.bStateConnectionToEnableFunctions := FALSE; END_IF
		IF NOT Lynus_Standards.GVL_Communicator.bStateConnectionToEnableFunctions THEN timDissableFunctions.IN := TRUE; ELSE timDissableFunctions.IN := FALSE; END_IF  
			timDissableFunctions(IN:= , PT:= Lynus_Standards.Constants_General.tTimeDissableLynusFunctions, Q=> , ET=> );
	
(*------------------------------------------------------------------Error----------------------------------------------------------------------------*)	

IF timDissableFunctions.Q THEN fbEHE.bWarning := TRUE; fbEHE.iWarningCode := 0; ELSE fbEHE.bWarning := FALSE; END_IF 
	IF (Lynus_Standards.GVL_Energy.stNumberOfDevices.diNumberOfEHE > Constants_Energy.diMaxNumberOfElectricHeatingElements) OR 
		(Lynus_Standards.GVL_Sensors.stDataTemperatureSensors[diNrOfTempS_IN].bEnabled AND Lynus_Standards.GVL_Sensors.stDataTemperatureSensors[diNrOfTempS_IN].byErrorWarning = 2) OR
			fbGetSystemTime.ERR THEN 
				fbEHE.bError := TRUE; 
	ELSE 
				fbEHE.bError := FALSE; 
	END_IF

IF Lynus_Standards.GVL_Energy.stNumberOfDevices.diNumberOfEHE > Constants_Energy.diMaxNumberOfElectricHeatingElements THEN fbEHE.iErrorCode := 1;
ELSIF fbGetSystemTime.ERR THEN fbEHE.iErrorCode := 3;
ELSIF Lynus_Standards.GVL_Sensors.stDataTemperatureSensors[diNrOfTempS_IN].bEnabled AND Lynus_Standards.GVL_Sensors.stDataTemperatureSensors[diNrOfTempS_IN].byErrorWarning = 2 THEN fbEHE.iErrorCode := 2;
END_IF  

(*------------------------------------------------------------------Logic----------------------------------------------------------------------------*)
	
//Calcualte the total SOC if we have more then 1 battery in our system
diNumberOfActiveBatterys := 0;
	dwSumSOC := 0;
		FOR liLPBatteryData := 1 TO Constants_Energy.diMaxNumberOfBatterys BY 1 DO
			IF Lynus_Standards.GVL_Energy.stDataOfBatterys[diNrOfEMS_IN,liLPBatteryData].bEnabled THEN diNumberOfActiveBatterys := diNumberOfActiveBatterys + 1; END_IF
				dwSumSOC := dwSumSOC + Lynus_Standards.GVL_Energy.stDataOfBatterys[diNrOfEMS_IN,liLPBatteryData].dwSOC;
		END_FOR
	
IF diNumberOfActiveBatterys > 0 THEN
	fbEHE.dwBatterySOC := DINT_TO_DWORD(DWORD_TO_DINT(dwSumSOC) / diNumberOfActiveBatterys);
ELSE
	fbEHE.dwBatterySOC := 100;	//When we have no battery in the ems system
END_IF

//Check if one or more Batterysystems or batteryinverter make island mode
diNumberOfBatteryInverterInEPO := 0;
	FOR liLPInEPO := 1 TO Constants_Energy.diMaxNumberOfBatteryInverters BY 1 DO
		IF Lynus_Standards.GVL_Energy.stDataOfBatteryInverters[diNrOfEMS_IN,liLPInEPO].bWorkOnIslandMode THEN fbEHE.bEPOIsActive := TRUE; diNumberOfBatteryInverterInEPO := diNumberOfBatteryInverterInEPO + 1; END_IF
	END_FOR 
		IF diNumberOfBatteryInverterInEPO <= 0 THEN fbEHE.bEPOIsActive := FALSE; END_IF

//Check the max. power of the grid connection and the sum of grid power
lrSizeGridConnection := 0;
	lrGridPower := 0;
		FOR liLPGridData := 1 TO Constants_Energy.diMaxNumberOfGridConnections BY 1 DO
			lrSizeGridConnection := lrSizeGridConnection + Lynus_Standards.GVL_Energy.stDataGridConnections[diNrOfEMS_IN,liLPGridData].rSizeGridConn;
				lrGridPower := lrGridPower + Lynus_Standards.GVL_Energy.stDataGridConnections[diNrOfEMS_IN,liLPGridData].lrPower;
		END_FOR	
	
//Digital input for external lock signal
fbDIExternalLock(bInvers:= FALSE, bSignal=> );

//Functionblock EHE
fbEHE(
	bEnable:= bEnable AND NOT timDissableFunctions.Q,
	bError:= , 
	bIsStepSwitched:= TRUE, 
	bEPOIsActive:= , 
	bExternalLock:= fbDIExternalLock.bSignal, 
	bWriteWithDelay:= TRUE,
	bTimeDissableFunctions:= timDissableFunctions.Q, 
	iErrorCode:= , 
	iWarningCode:= , 
	diNumberOfEHE:= diNrOfEHE_OUT,
	dwBatterySOC:= ,
	lrSizeGridConnection:= lrSizeGridConnection,
	lrGridPower:= lrGridPower, 
	lrTotalCounterEnergy_Consumption:= , 
	lrTotalCounterEnergy_Production:= , 
	lrCounterEnergyT1_Consumption:= , 
	lrCounterEnergyT2_Consumption:= , 
	lrCounterEnergyT1_Production:= , 
	lrCounterEnergyT2_Production:= , 
	lrPowerEHE:= , 
	arrTargetPower:= Lynus_Standards.GVL_Energy.stDataElectricHeatingElements[diNrOfEMS_IN,diNrOfEHE_OUT].arrTargetPowerEMS, 
	rTemperatureInBoiler:= Lynus_Standards.GVL_Sensors.stDataTemperatureSensors[diNrOfTempS_IN].rTemperature, 
	tTimDelayOutput:= T#5S, 
	stSystemTime:= , 
	stSetupEHE:= stSetupEHE, 
	stDataEHEOut=> , 
	stDataEHEOutDelay=> stDataEHE);

//Target Power, to use this on a external Function
rTargetPowerForExtFunc := fbEHE.stDataEHEOut.rTargetPower;
	
(*-------------------------------------------------------------------------Output----------------------------------------------------------------------*)

fbAOEHE(
	rYMinTerminalValue:= 0, 
	rXMinInputSignal:= 0, 
	rYMaxTerminalValue:= 32767, 
	rXMaxInputSignal:= 100, 
	rSignal:= fbEHE.stDataEHEOut.rTargetPower, 
	usiState=> );

(*-----------------------------------------------------------Handle data to Global structure for the electric heating element-----------------------------------------------------------------*)

//Delte al old Data on GVL after a online change or change on the variable diNrOfEMS_IDOD
IF diNrOfEMS_IN <> diNrOfEMS_IN_CP AND iStateGVLData = 0 THEN iStateGVLData := 10; END_IF 

CASE iStateGVLData OF
	
	0://Init Step
		byWaitInStep := 0;
			diCounterForGVL := 1;
	
	1://Wait for 4 Steps before clean al Data on GVL
		byWaitInStep := byWaitInStep + 1;
			IF byWaitInStep >= 4 AND fbNumberDevice.bNumberIsCalculatet THEN iStateGVLData := 2; END_IF
				//To much Devices, back to the Init step
				IF byWaitInStep >= 4 AND NOT fbNumberDevice.bNumberIsCalculatet THEN iStateGVLData := 0; END_IF	
			
	2://Clear all Data in GVL
		FOR diLPForGVL := 1 TO Constants_Energy.diMaxNumberOfEMS BY 1 DO 
			Lynus_Standards.GVL_Energy.stDataElectricHeatingElements[diLPForGVL,diCounterForGVL].bEnabled := FALSE;
				Lynus_Standards.GVL_Energy.stDataElectricHeatingElements[diLPForGVL,diCounterForGVL].bIsStepSwitched := FALSE;
					Lynus_Standards.GVL_Energy.stDataElectricHeatingElements[diLPForGVL,diCounterForGVL].bIsControllable := FALSE;
						Lynus_Standards.GVL_Energy.stDataElectricHeatingElements[diLPForGVL,diCounterForGVL].byPriority := 0;
							Lynus_Standards.GVL_Energy.stDataElectricHeatingElements[diLPForGVL,diCounterForGVL].byErrorWarning := 0;
								Lynus_Standards.GVL_Energy.stDataElectricHeatingElements[diLPForGVL,diCounterForGVL].byNumberOfSteps := 0;
									Lynus_Standards.GVL_Energy.stDataElectricHeatingElements[diLPForGVL,diCounterForGVL].lrPower := 0;
										Lynus_Standards.GVL_Energy.stDataElectricHeatingElements[diLPForGVL,diCounterForGVL].lrPowerConsumption := 0;
											Lynus_Standards.GVL_Energy.stDataElectricHeatingElements[diLPForGVL,diCounterForGVL].lrPowerProduction := 0;
												FOR byLPGVLSetMaxPower := 1 TO 10 BY 1 DO
													Lynus_Standards.GVL_Energy.stDataElectricHeatingElements[diLPForGVL,diCounterForGVL].arrMaxPower[byLPGVLSetMaxPower] := 0;
												END_FOR 
													//Set also the target value from ems back here to 0 and not in EMS function because EMS is in Standy when we have a online change (Problem when we delete a ems function and make a online change)
													FOR byLPGVLSetMaxPower := 1 TO 10 BY 1 DO
														Lynus_Standards.GVL_Energy.stDataElectricHeatingElements[diLPForGVL,diCounterForGVL].arrTargetPowerEMS[byLPGVLSetMaxPower] := 0;	
													END_FOR
		END_FOR
			diCounterForGVL := diCounterForGVL + 1;
				diCounterForGVL := LIMIT(0,diCounterForGVL,Constants_Energy.diMaxNumberOfElectricHeatingElements);
					//Back to the init step
					IF diCounterForGVL >= Constants_Energy.diMaxNumberOfElectricHeatingElements THEN iStateGVLData := 0; END_IF

	10://Clear old Data on GVL 	
		Lynus_Standards.GVL_Energy.stDataElectricHeatingElements[diNrOfEMS_IN_CP,diNrOfEHE_OUT].bEnabled := FALSE;
			Lynus_Standards.GVL_Energy.stDataElectricHeatingElements[diNrOfEMS_IN_CP,diNrOfEHE_OUT].bIsStepSwitched := FALSE;
				Lynus_Standards.GVL_Energy.stDataElectricHeatingElements[diNrOfEMS_IN_CP,diNrOfEHE_OUT].bIsControllable := FALSE;
					Lynus_Standards.GVL_Energy.stDataElectricHeatingElements[diNrOfEMS_IN_CP,diNrOfEHE_OUT].byPriority := 0;
						Lynus_Standards.GVL_Energy.stDataElectricHeatingElements[diNrOfEMS_IN_CP,diNrOfEHE_OUT].byErrorWarning := 0;
							Lynus_Standards.GVL_Energy.stDataElectricHeatingElements[diNrOfEMS_IN_CP,diNrOfEHE_OUT].byNumberOfSteps := 0;
								Lynus_Standards.GVL_Energy.stDataElectricHeatingElements[diNrOfEMS_IN_CP,diNrOfEHE_OUT].lrPower := 0;
									Lynus_Standards.GVL_Energy.stDataElectricHeatingElements[diNrOfEMS_IN_CP,diNrOfEHE_OUT].lrPowerConsumption := 0;
										Lynus_Standards.GVL_Energy.stDataElectricHeatingElements[diNrOfEMS_IN_CP,diNrOfEHE_OUT].lrPowerProduction := 0;
											FOR byLPGVLSetMaxPower := 1 TO 10 BY 1 DO
												Lynus_Standards.GVL_Energy.stDataElectricHeatingElements[diNrOfEMS_IN_CP,diNrOfEHE_OUT].arrMaxPower[byLPGVLSetMaxPower] := 0;
											END_FOR 
												
		diNrOfEMS_IN_CP := diNrOfEMS_IN;
			//Back to the init step
			iStateGVLData := 0;

END_CASE 	 

IF diNrOfEHE_OUT > 0 AND fbNumberDevice.bNumberIsCalculatet AND diNrOfEMS_IN > 0 THEN
	Lynus_Standards.GVL_Energy.stDataElectricHeatingElements[diNrOfEMS_IN,diNrOfEHE_OUT].bEnabled := fbEHE.stDataEHEOut.bEnabled;
		Lynus_Standards.GVL_Energy.stDataElectricHeatingElements[diNrOfEMS_IN,diNrOfEHE_OUT].bIsStepSwitched := fbEHE.stDataEHEOut.bIsStepSwitched;
			Lynus_Standards.GVL_Energy.stDataElectricHeatingElements[diNrOfEMS_IN,diNrOfEHE_OUT].bIsControllable := TRUE;
				Lynus_Standards.GVL_Energy.stDataElectricHeatingElements[diNrOfEMS_IN,diNrOfEHE_OUT].byPriority := fbEHE.stDataEHEOut.byPriority;
					Lynus_Standards.GVL_Energy.stDataElectricHeatingElements[diNrOfEMS_IN,diNrOfEHE_OUT].byErrorWarning := fbEHE.stDataEHEOut.byErrorWarning;
						Lynus_Standards.GVL_Energy.stDataElectricHeatingElements[diNrOfEMS_IN,diNrOfEHE_OUT].byNumberOfSteps := fbEHE.stDataEHEOut.byNumberOfSteps;
							Lynus_Standards.GVL_Energy.stDataElectricHeatingElements[diNrOfEMS_IN,diNrOfEHE_OUT].lrPower := fbEHE.stDataEHEOut.lrPower;
								Lynus_Standards.GVL_Energy.stDataElectricHeatingElements[diNrOfEMS_IN,diNrOfEHE_OUT].lrPowerConsumption := fbEHE.stDataEHEOut.lrPowerConsumption;
									Lynus_Standards.GVL_Energy.stDataElectricHeatingElements[diNrOfEMS_IN,diNrOfEHE_OUT].lrPowerProduction := fbEHE.stDataEHEOut.lrPowerProduction;
										Lynus_Standards.GVL_Energy.stDataElectricHeatingElements[diNrOfEMS_IN,diNrOfEHE_OUT].arrMaxPower := fbEHE.stDataEHEOut.arrMaxPower; 
END_IF				

(*----------------------------------------------------------Save persistent data----------------------------------------------------------------*)

arrPD[1](lrValue:= BOOL_TO_LREAL(bEnable), bEventBasedActive=> );
arrPD[2](lrValue:= BOOL_TO_LREAL(bPowerDataInvers), bEventBasedActive=> );
arrPD[3](lrValue:= DINT_TO_LREAL(diNrOfEMS_IN), bEventBasedActive=> );
arrPD[4](lrValue:= DINT_TO_LREAL(diNrOfEM_IN_EHE), bEventBasedActive=> );
arrPD[5](lrValue:= DINT_TO_LREAL(diNrOfTempS_IN), bEventBasedActive=> );
arrPD[6](lrValue:= REAL_TO_LREAL(stSetupEHE.rMaxPower1), bEventBasedActive=> );
arrPD[7](lrValue:= REAL_TO_LREAL(stSetupEHE.rMaxPower2), bEventBasedActive=> );
arrPD[8](lrValue:= REAL_TO_LREAL(stSetupEHE.rMaxPower3), bEventBasedActive=> );
arrPD[9](lrValue:= REAL_TO_LREAL(stSetupEHE.rMaxPower4), bEventBasedActive=> );
arrPD[10](lrValue:= REAL_TO_LREAL(stSetupEHE.rMaxPower5), bEventBasedActive=> );
arrPD[11](lrValue:= REAL_TO_LREAL(stSetupEHE.rMaxPower6), bEventBasedActive=> );
arrPD[12](lrValue:= REAL_TO_LREAL(stSetupEHE.rMaxPower7), bEventBasedActive=> );
arrPD[13](lrValue:= REAL_TO_LREAL(stSetupEHE.rMaxPower8), bEventBasedActive=> );
arrPD[14](lrValue:= REAL_TO_LREAL(stSetupEHE.rMaxPower9), bEventBasedActive=> );
arrPD[15](lrValue:= REAL_TO_LREAL(stSetupEHE.rMaxPower10), bEventBasedActive=> );
arrPD[16](lrValue:= BOOL_TO_LREAL(stSetupEHE.bDisableLegionellaPr), bEventBasedActive=> );
arrPD[17](lrValue:= BOOL_TO_LREAL(stSetupEHE.bManualyOn), bEventBasedActive=> );
arrPD[18](lrValue:= BOOL_TO_LREAL(stSetupEHE.bOnEmergPowerOff), bEventBasedActive=> );
arrPD[19](lrValue:= BOOL_TO_LREAL(stSetupEHE.bTimeEnabled), bEventBasedActive=> );
arrPD[20](lrValue:= BYTE_TO_LREAL(stSetupEHE.byDisableSOC), bEventBasedActive=> );
arrPD[21](lrValue:= BYTE_TO_LREAL(stSetupEHE.byEnableSOC), bEventBasedActive=> );
arrPD[22](lrValue:= BYTE_TO_LREAL(stSetupEHE.byHourOff), bEventBasedActive=> );
arrPD[23](lrValue:= BYTE_TO_LREAL(stSetupEHE.byHourOn), bEventBasedActive=> );
arrPD[24](lrValue:= BYTE_TO_LREAL(stSetupEHE.byManualyTargetPower), bEventBasedActive=> );
arrPD[25](lrValue:= BYTE_TO_LREAL(stSetupEHE.byMinutesOff), bEventBasedActive=> );
arrPD[26](lrValue:= BYTE_TO_LREAL(stSetupEHE.byMinutesOn), bEventBasedActive=> );
arrPD[27](lrValue:= BYTE_TO_LREAL(stSetupEHE.byPriority), bEventBasedActive=> );
arrPD[28](lrValue:= UINT_TO_LREAL(stSetupEHE.uiTargetTempMax), bEventBasedActive=> );
arrPD[29](lrValue:= UINT_TO_LREAL(stSetupEHE.uiTargetTempOff), bEventBasedActive=> );
arrPD[30](lrValue:= UINT_TO_LREAL(stSetupEHE.uiTargetTempOn), bEventBasedActive=> );
arrPD[31](lrValue:= DINT_TO_LREAL(diNrOfEMS_IN_CP), bEventBasedActive=> );

END_FUNCTION_BLOCK

// ---- FBs/Generator/FB_Generator_OnOff.TcPOU
FUNCTION_BLOCK FB_Generator_OnOff
VAR_INPUT PERSISTENT
	bEnable									: BOOL;															//{#lynus.ag#()} //Enable the Fuctionblock and his logic
	bPowerDataInvers						: BOOL;															//With True its possible to invert all received power data from the electric meter
	diNrOfEMS_IN							: DINT;															//Number of EMS what control this Device.
	diNrOfEM_IN_Generator					: DINT;															//Number of the electric meter for incoming power data. (Power Data for this Device)
	stSetupGenerator						: ST_Setup_Generator;											//{#lynus.ag#()} //Setup Generator
END_VAR
VAR_INPUT
END_VAR
VAR_OUTPUT
	stDataGenerator							: ST_Generator_Output;											//{#lynus.ag#()} //Generator output data
	diNrOfGenerator_OUT						: DINT;															//Active Number from the Gnerator for using on other functions
END_VAR		
VAR
	{attribute 'hide'}
	fbGenerator								: FB_Generator;													//Fb Generator
	{attribute 'hide'}
	fbNumberDevice							: FB_NumberOfDevice;											//Function block to calcualte the number of the Device
	fbDIErrorGenerator						: FB_XL1XXX_DI;													//Digital Input Error Generator
	fbDOStartGenerator						: FB_XL2XXX_DO;													//Digital output start generator
	fbDOResetGenerator						: FB_XL2XXX_DO;													//Digital output to reset the generator after a error
	{attribute 'hide'}
	timDissableFunctions					: TON;															//Timer to dissable the Function after Lynus_Standards.Constants_General.tTimeDissableLynusFunctions Days without connection to the Lynus Cloud
	{attribute 'hide'}
	timResetConnectionOnGVL					: TON;															//Timer to try reset the connection Flag on the GVL. (When somebody delete the Connection Function and make only a onlinechange)
	{attribute 'hide'}
	FNReset									: F_TRIG;														//Reset Generator
	{attribute 'hide'}
	arrSOC									: ARRAY[1..Constants_Energy.diMaxNumberOfBatterys] OF DWORD;	//Array with al SOC from all batterys in this ems function
	{attribute 'hide'}
	arrPD									: ARRAY[1..6] OF FB_PersistentData_Number;						//Function to save persistent data 
	{attribute 'hide'}
	byWaitInStep							: BYTE;															//Wait in Step before start to clean data on PLC
	{attribute 'hide'}
	iStateGVLData							: INT;															//State machine to handle the data on the GVL
	{attribute 'hide'}
	diNumberOfActiveBatterys				: DINT;															//Number of active batterys
	{attribute 'hide'}
	diCounterForGVL							: DINT;															//Counter to clean old data on GVL
	{attribute 'hide'}
	dwSumSOC								: DWORD;														//Sum of the SOC from all batterys
	{attribute 'hide'}
	liLPBatteryData							: LINT;															//Loop to check some data from batterys
	{attribute 'hide'}
	liLPBattSOC100							: LINT;															//Loop to ckeck if some battery has the soc value >= 0	
END_VAR

//Creator : Kai Ebensperger
//Company : Lynus AG
//Date : 07.06.2021
//Version : 1.0.0.0

//With this function is possible to control a generator with digital Inputs and Outputs from the plc
//With the Nr from the Electric Meter its possible to send the data fromt the electric meter directly to the Generator function to display it

//NOTE for diNr.....Designation => 
//_IN = Here Data come in from other Functions or go out to other functions about the GVL
//_OUT = Here Data go out to other functions about the GVL

(*------------------------------------------------------------Limits----------------------------------------------------------------------------------*)

diNrOfEMS_IN := LIMIT(0,diNrOfEMS_IN,Constants_Energy.diMaxNumberOfEMS);
	diNrOfEM_IN_Generator := LIMIT(0,diNrOfEM_IN_Generator,Constants_Energy.diMaxNumberOfElectricMeters);	

(*------------------------------------------------------------------Power Data----------------------------------------------------------------------------*)

IF NOT bPowerDataInvers THEN
	fbGenerator.lrCounterEnergyT1_Consumption := Lynus_Standards.GVL_Energy.stDataElectricMeters[diNrOfEM_IN_Generator].lrCounterEnergyT1_Production * 1000;
	fbGenerator.lrCounterEnergyT2_Consumption := Lynus_Standards.GVL_Energy.stDataElectricMeters[diNrOfEM_IN_Generator].lrCounterEnergyT2_Production * 1000;
	fbGenerator.lrCounterEnergyT1_Production := Lynus_Standards.GVL_Energy.stDataElectricMeters[diNrOfEM_IN_Generator].lrCounterEnergyT1_Consumption * 1000;
	fbGenerator.lrCounterEnergyT2_Production := Lynus_Standards.GVL_Energy.stDataElectricMeters[diNrOfEM_IN_Generator].lrCounterEnergyT1_Consumption * 1000;
	fbGenerator.lrTotalCounterEnergy_Consumption := Lynus_Standards.GVL_Energy.stDataElectricMeters[diNrOfEM_IN_Generator].lrTotalCounterEnergy_Production * 1000;
	fbGenerator.lrTotalCounterEnergy_Production := Lynus_Standards.GVL_Energy.stDataElectricMeters[diNrOfEM_IN_Generator].lrTotalCounterEnergy_Consumption * 1000;
ELSE
	fbGenerator.lrCounterEnergyT1_Consumption := Lynus_Standards.GVL_Energy.stDataElectricMeters[diNrOfEM_IN_Generator].lrCounterEnergyT1_Consumption * 1000;
	fbGenerator.lrCounterEnergyT2_Consumption := Lynus_Standards.GVL_Energy.stDataElectricMeters[diNrOfEM_IN_Generator].lrCounterEnergyT2_Consumption * 1000;
	fbGenerator.lrCounterEnergyT1_Production := Lynus_Standards.GVL_Energy.stDataElectricMeters[diNrOfEM_IN_Generator].lrCounterEnergyT1_Production * 1000;
	fbGenerator.lrCounterEnergyT2_Production := Lynus_Standards.GVL_Energy.stDataElectricMeters[diNrOfEM_IN_Generator].lrCounterEnergyT2_Production * 1000;
	fbGenerator.lrTotalCounterEnergy_Consumption := Lynus_Standards.GVL_Energy.stDataElectricMeters[diNrOfEM_IN_Generator].lrTotalCounterEnergy_Consumption * 1000;
	fbGenerator.lrTotalCounterEnergy_Production := Lynus_Standards.GVL_Energy.stDataElectricMeters[diNrOfEM_IN_Generator].lrTotalCounterEnergy_Production * 1000;
END_IF	
	
(*-------------------------------------------------------------Calcualte the number of Generator---------------------------------------------------------------*)

fbNumberDevice(
	diActualNumberOfDevices:= Lynus_Standards.GVL_Energy.stNumberOfDevices.diNumberOfGenerators, 
	diMaxNumberOfDevices:= Constants_Energy.diMaxNumberOfGenerators, 
	udiCounterOnlineChange:= TwinCAT_SystemInfoVarList._AppInfo.OnlineChangeCnt, 
	bNumberIsCalculatet=> , 
	bFPNumberIsCalculatet=> , 
	bOnlineChange=> , 
	diNumberForThisDevice=> diNrOfGenerator_OUT, 
	diNumberOfTotalDevices=> );

//Write new Numer on GVL
IF fbNumberDevice.bFPNumberIsCalculatet THEN
	Lynus_Standards.GVL_Energy.stNumberOfDevices.diNumberOfGenerators := fbNumberDevice.diNumberOfTotalDevices;	
END_IF 

//Delete old Number on GVL
IF fbNumberDevice.bOnlineChange THEN 
	Lynus_Standards.GVL_Energy.stNumberOfDevices.diNumberOfGenerators := diNrOfGenerator_OUT;	
		iStateGVLData := 1; 
END_IF
			
(*------------------------------------------------------------------FB Generator----------------------------------------------------------------------------*)

//Calcualte the total SOC if we have more then 1 battery in our system
diNumberOfActiveBatterys := 0;
	dwSumSOC := 0;
		FOR liLPBatteryData := 1 TO Constants_Energy.diMaxNumberOfBatterys BY 1 DO
			IF Lynus_Standards.GVL_Energy.stDataOfBatterys[diNrOfEMS_IN,liLPBatteryData].bEnabled THEN diNumberOfActiveBatterys := diNumberOfActiveBatterys + 1; END_IF
				dwSumSOC := dwSumSOC + Lynus_Standards.GVL_Energy.stDataOfBatterys[diNrOfEMS_IN,liLPBatteryData].dwSOC;
					arrSOC[liLPBatteryData] := Lynus_Standards.GVL_Energy.stDataOfBatterys[diNrOfEMS_IN,liLPBatteryData].dwSOC; 
		END_FOR

IF diNumberOfActiveBatterys > 0 THEN
	fbGenerator.dwBatterySOC := DINT_TO_DWORD(DWORD_TO_DINT(dwSumSOC) / diNumberOfActiveBatterys);
END_IF

//If we have more then 1 battery in system switch off when 1 battery has reached the value 100 to not overload the batterysystem
FOR liLPBattSOC100 := 1 TO Constants_Energy.diMaxNumberOfBatterys BY 1 DO
	IF arrSOC[liLPBattSOC100] >= 100 THEN fbGenerator.dwBatterySOC := 100; END_IF
END_FOR 

(*-------------------------------------------------------------Service from Backend is ready and check the connection to backen for dissabel/enable Function---------------------------------------------------------------*)

//Try to reset the variable for connection on the GVL. When all is normal then the Lynus Mqtt connection function set this variable to true in the next cycle
//When we have no connection to the backend then after Lynus_Standards.Constants_General.tTimeDissableLynusFunctions days the Function is dissabled with all of his functionalities
timResetConnectionOnGVL(IN:= NOT timResetConnectionOnGVL.Q, PT:= T#1H, Q=> , ET=> );
	IF timResetConnectionOnGVL.Q THEN Lynus_Standards.GVL_Communicator.bStateConnectionToEnableFunctions := FALSE; END_IF
		IF NOT Lynus_Standards.GVL_Communicator.bStateConnectionToEnableFunctions THEN timDissableFunctions.IN := TRUE; ELSE timDissableFunctions.IN := FALSE; END_IF  
			timDissableFunctions(IN:= , PT:= Lynus_Standards.Constants_General.tTimeDissableLynusFunctions, Q=> , ET=> );

(*-----------------------------------------------------------------------------Error and Reset----------------------------------------------------------------------------*)

fbDIErrorGenerator(bInvers:= FALSE, bSignal=> );

IF timDissableFunctions.Q THEN fbGenerator.bWarning := TRUE; fbGenerator.iWarningCode := 0; ELSE fbGenerator.bWarning := FALSE; END_IF 
	IF fbDIErrorGenerator.bSignal OR Lynus_Standards.GVL_Energy.stNumberOfDevices.diNumberOfGenerators > Constants_Energy.diMaxNumberOfGenerators THEN fbGenerator.bError := TRUE; ELSE fbGenerator.bError := FALSE; END_IF 

IF Lynus_Standards.GVL_Energy.stNumberOfDevices.diNumberOfGenerators > Constants_Energy.diMaxNumberOfGenerators THEN fbGenerator.iErrorCode := 1;
ELSIF fbDIErrorGenerator.bSignal THEN fbGenerator.iErrorCode := 0;
END_IF  

FNReset(CLK:= fbGenerator.stDataGeneratorOut.bSReset, Q=> );

fbGenerator(
	bEnable:= bEnable AND NOT timDissableFunctions.Q,
	bError:= , 
	bReset:= FNReset.Q,  
	bWriteWithDelay:= TRUE, 
	iErrorCode:= , 
	iWarningCode:= , 
	dwBatterySOC:= , 
	lrTotalCounterEnergy_Consumption:= , 
	lrTotalCounterEnergy_Production:= , 
	lrCounterEnergyT1_Consumption:= , 
	lrCounterEnergyT2_Consumption:= , 
	lrCounterEnergyT1_Production:= , 
	lrCounterEnergyT2_Production:= , 
	lrPowerGenerator:= Lynus_Standards.GVL_Energy.stDataElectricMeters[diNrOfEM_IN_Generator].lrPower * 1000, 
	tDelaySwitchOn:= T#15S, 
	tTimDelayOutput:= T#5S, 
	stSetupGenerator:= stSetupGenerator, 
	stDataGeneratorOut=> , 
	stDataGeneratorOutDelay=> stDataGenerator);
	
(*-------------------------------------------------------------------------Output----------------------------------------------------------------------*)

fbDOStartGenerator(bInvers:= FALSE, bSignal:= fbGenerator.stDataGeneratorOut.bOutput);
	fbDOResetGenerator(bInvers:= FALSE, bSignal:= fbGenerator.stDataGeneratorOut.bSReset);
	
(*-----------------------------------------------------------Handle data to Global structure for the Generator system-----------------------------------------------------------------*)

CASE iStateGVLData OF
	
	0://Init Step
		byWaitInStep := 0;
			diCounterForGVL := 1;
	
	1://Wait for 4 Steps before clean al Data on GVL
		byWaitInStep := byWaitInStep + 1;
			IF byWaitInStep >= 4 AND fbNumberDevice.bNumberIsCalculatet THEN iStateGVLData := 2; END_IF
				//To much Devices, back to the Init step
				IF byWaitInStep >= 4 AND NOT fbNumberDevice.bNumberIsCalculatet THEN iStateGVLData := 0; END_IF	
			
	2://Clear all Data in GVL
		Lynus_Standards.GVL_Energy.stDataOfGenerators[diCounterForGVL].bEnabled := FALSE;
			Lynus_Standards.GVL_Energy.stDataOfGenerators[diCounterForGVL].bOutput := FALSE;
				Lynus_Standards.GVL_Energy.stDataOfGenerators[diCounterForGVL].bSReset := 0;
					Lynus_Standards.GVL_Energy.stDataOfGenerators[diCounterForGVL].byErrorWarning := 0;
						Lynus_Standards.GVL_Energy.stDataOfGenerators[diCounterForGVL].lrPowerConsumption := 0;
							Lynus_Standards.GVL_Energy.stDataOfGenerators[diCounterForGVL].lrPower := 0;
								Lynus_Standards.GVL_Energy.stDataOfGenerators[diCounterForGVL].lrPowerProduction := 0;
		
		diCounterForGVL := diCounterForGVL + 1;
			diCounterForGVL := LIMIT(0,diCounterForGVL,Constants_Energy.diMaxNumberOfGenerators);
				//Back to the init step
				IF diCounterForGVL >= Constants_Energy.diMaxNumberOfGenerators THEN iStateGVLData := 0; END_IF

END_CASE 	 

IF diNrOfGenerator_OUT > 0 AND fbNumberDevice.bNumberIsCalculatet THEN
	Lynus_Standards.GVL_Energy.stDataOfGenerators[diNrOfGenerator_OUT].bEnabled := fbGenerator.stDataGeneratorOut.bEnabled;
		Lynus_Standards.GVL_Energy.stDataOfGenerators[diNrOfGenerator_OUT].bOutput := fbGenerator.stDataGeneratorOut.bOutput;
			Lynus_Standards.GVL_Energy.stDataOfGenerators[diNrOfGenerator_OUT].bSReset := fbGenerator.stDataGeneratorOut.bSReset;
				Lynus_Standards.GVL_Energy.stDataOfGenerators[diNrOfGenerator_OUT].byErrorWarning := fbGenerator.stDataGeneratorOut.byErrorWarning;
					Lynus_Standards.GVL_Energy.stDataOfGenerators[diNrOfGenerator_OUT].lrPowerConsumption := fbGenerator.stDataGeneratorOut.lrPowerConsumption;
						Lynus_Standards.GVL_Energy.stDataOfGenerators[diNrOfGenerator_OUT].lrPower := fbGenerator.stDataGeneratorOut.lrPower;
							Lynus_Standards.GVL_Energy.stDataOfGenerators[diNrOfGenerator_OUT].lrPowerProduction := fbGenerator.stDataGeneratorOut.lrPowerProduction;	
END_IF 				

(*----------------------------------------------------------Save persistent data----------------------------------------------------------------*)

arrPD[1](lrValue:= BOOL_TO_LREAL(bEnable), bEventBasedActive=> );
arrPD[2](lrValue:= BOOL_TO_LREAL(bPowerDataInvers), bEventBasedActive=> );
arrPD[3](lrValue:= DINT_TO_LREAL(diNrOfEMS_IN), bEventBasedActive=> );
arrPD[4](lrValue:= DINT_TO_LREAL(diNrOfEM_IN_Generator), bEventBasedActive=> );
arrPD[5](lrValue:= BYTE_TO_LREAL(stSetupGenerator.byDisableSOC), bEventBasedActive=> );
arrPD[6](lrValue:= BYTE_TO_LREAL(stSetupGenerator.byEnableSOC), bEventBasedActive=> );

END_FUNCTION_BLOCK

// ---- FBs/Grid/FB_Grid_Power.TcPOU
FUNCTION_BLOCK FB_Grid_Power
VAR_INPUT PERSISTENT
	bEnable									: BOOL;													//Enable the Fuctionblock and his logic
	diNrOfEMS_IN							: DINT;													//Number of EMS on what this Device send Data
	diNrOfEM_IN_Grid						: DINT;													//Number of the electric meter for incoming power data. (Power Data for this Device)
	rSizeGridConn							: REAL;													//{#lynus.ag#()} //Max Size of the Grid connection in kW
END_VAR
VAR_INPUT
END_VAR
VAR_OUTPUT
	stDataGrid								: ST_GridConnection_Output;								//{#lynus.ag#()} //Output Data from the Grid
	diNrOfGrid_OUT							: DINT;													//Active Number from the Grid connection for using on other functions
END_VAR
VAR
	{attribute 'hide'}
	fbGrid									: FB_GridConnection;									//Function block for grid connection
	{attribute 'hide'}
	fbNumberDevice							: FB_NumberOfDevice;									//Function block to calcualte the number of the Device
	{attribute 'hide'}
	timDissableFunctions					: TON;													//Timer to dissable the Function after Lynus_Standards.Constants_General.tTimeDissableLynusFunctions Days without connection to the Lynus Cloud
	{attribute 'hide'}	
	timResetConnectionOnGVL					: TON;													//Timer to try reset the connection Flag on the GVL. (When somebody delete the Connection Function and make only a onlinechange)
	{attribute 'hide'}
	arrPD									: ARRAY[1..5] OF FB_PersistentData_Number;				//Function to save persistent data 
	{attribute 'hide'}
	byWaitInStep							: BYTE;													//Wait in Step before start to clean data on PLC
	{attribute 'hide'}
	iStateGVLData							: INT;													//State machine to handle the data on the GVL
	{attribute 'hide'}
	diCounterForGVL							: DINT;													//Counter to clean old data on GVL
	{attribute 'hide'}
	diLPForGVL								: DINT;													//Loop to clean old data on GVL
END_VAR
VAR PERSISTENT
	{attribute 'conditionalshow'}
	diNrOfEMS_IN_CP							: DINT;													//Number of EMS what control this Device to compare with the original
END_VAR

//Creator : Kai Ebensperger
//Company : Lynus AG
//Date : 07.06.2021
//Version : 1.0.0.0

//With this function block its possible to show the power data from a grid connection.
//The size from the Grid connection is sending to the ems

//NOTE for diNr.....Designation => 
//_IN = Here Data come in from other Functions or go out to other functions about the GVL
//_OUT = Here Data go out to other functions about the GVL

(*------------------------------------------------------------Limits----------------------------------------------------------------------------------*)

diNrOfEMS_IN := LIMIT(0,diNrOfEMS_IN,Constants_Energy.diMaxNumberOfEMS);
	diNrOfEM_IN_Grid := LIMIT(0,diNrOfEM_IN_Grid,Constants_Energy.diMaxNumberOfElectricMeters);

(*-------------------------------------------------------------Calcualte the number of Grid connection---------------------------------------------------------------*)

fbNumberDevice(
	diActualNumberOfDevices:= Lynus_Standards.GVL_Energy.stNumberOfDevices.diNumberOfGrids, 
	diMaxNumberOfDevices:= Constants_Energy.diMaxNumberOfGridConnections, 
	udiCounterOnlineChange:= TwinCAT_SystemInfoVarList._AppInfo.OnlineChangeCnt, 
	bNumberIsCalculatet=> , 
	bFPNumberIsCalculatet=> , 
	bOnlineChange=> , 
	diNumberForThisDevice=> diNrOfGrid_OUT, 
	diNumberOfTotalDevices=> );

//Write new Numer on GVL
IF fbNumberDevice.bFPNumberIsCalculatet THEN
	Lynus_Standards.GVL_Energy.stNumberOfDevices.diNumberOfGrids := fbNumberDevice.diNumberOfTotalDevices;	
END_IF 

//Delete old Number on GVL
IF fbNumberDevice.bOnlineChange THEN 
	Lynus_Standards.GVL_Energy.stNumberOfDevices.diNumberOfGrids := diNrOfGrid_OUT;	
		iStateGVLData := 1; 
END_IF	

(*-------------------------------------------------------------Service from Backend is ready and check the connection to backen for dissabel/enable Function---------------------------------------------------------------*)

//Try to reset the variable for connection on the GVL. When all is normal then the Lynus Mqtt connection function set this variable to true in the next cycle
//When we have no connection to the backend then after Lynus_Standards.Constants_General.tTimeDissableLynusFunctions days the Function is dissabled with all of his functionalities
timResetConnectionOnGVL(IN:= NOT timResetConnectionOnGVL.Q, PT:= T#1H, Q=> , ET=> );
	IF timResetConnectionOnGVL.Q THEN Lynus_Standards.GVL_Communicator.bStateConnectionToEnableFunctions := FALSE; END_IF
		IF NOT Lynus_Standards.GVL_Communicator.bStateConnectionToEnableFunctions THEN timDissableFunctions.IN := TRUE; ELSE timDissableFunctions.IN := FALSE; END_IF  
			timDissableFunctions(IN:= , PT:= Lynus_Standards.Constants_General.tTimeDissableLynusFunctions, Q=> , ET=> );

(*------------------------------------------------------------------Error----------------------------------------------------------------------------*)

IF timDissableFunctions.Q THEN fbGrid.bWarning := TRUE; fbGrid.iWarningCode := 0; ELSE fbGrid.bWarning := FALSE; END_IF 			
	IF Lynus_Standards.GVL_Energy.stDataElectricMeters[diNrOfEM_IN_Grid].byErrorWarning = 2 OR Lynus_Standards.GVL_Energy.stNumberOfDevices.diNumberOfGrids > Constants_Energy.diMaxNumberOfGridConnections THEN fbGrid.bError := TRUE; ELSE fbGrid.bError := FALSE; END_IF 

IF Lynus_Standards.GVL_Energy.stNumberOfDevices.diNumberOfGrids > Constants_Energy.diMaxNumberOfGridConnections THEN fbGrid.iErrorCode := 1;
ELSIF Lynus_Standards.GVL_Energy.stDataElectricMeters[diNrOfEM_IN_Grid].byErrorWarning = 2 THEN fbGrid.iErrorCode := 0;
END_IF  

(*------------------------------------------------------------------FB Grid----------------------------------------------------------------------------*)

fbGrid(
	bEnable:= bEnable AND NOT timDissableFunctions.Q, 
	bError:= , 
	bWriteWithDelay:= TRUE, 
	iErrorCode:= , 
	iWarningCode:= , 
	lrTotalCounterEnergy_Consumption:= Lynus_Standards.GVL_Energy.stDataElectricMeters[diNrOfEM_IN_Grid].lrTotalCounterEnergy_Consumption * 1000, 
	lrTotalCounterEnergy_Production:= Lynus_Standards.GVL_Energy.stDataElectricMeters[diNrOfEM_IN_Grid].lrTotalCounterEnergy_Production * 1000, 
	lrCounterEnergyT1_Consumption:= Lynus_Standards.GVL_Energy.stDataElectricMeters[diNrOfEM_IN_Grid].lrCounterEnergyT1_Consumption * 1000, 
	lrCounterEnergyT2_Consumption:= Lynus_Standards.GVL_Energy.stDataElectricMeters[diNrOfEM_IN_Grid].lrCounterEnergyT2_Consumption * 1000, 
	lrCounterEnergyT1_Production:= Lynus_Standards.GVL_Energy.stDataElectricMeters[diNrOfEM_IN_Grid].lrCounterEnergyT1_Production * 1000, 
	lrCounterEnergyT2_Production:= Lynus_Standards.GVL_Energy.stDataElectricMeters[diNrOfEM_IN_Grid].lrCounterEnergyT2_Production * 1000, 
	lrPowerGrid:= Lynus_Standards.GVL_Energy.stDataElectricMeters[diNrOfEM_IN_Grid].lrPower * 1000, 
	rSizeGridConn:= rSizeGridConn, 
	tTimDelayOutput:= T#5S, 
	stDataGridOut=> , 
	stDataGridOutDelay=> stDataGrid);
	
(*-----------------------------------------------------------Handle data to Global structure for the grid connections-----------------------------------------------------------------*)

//Delte al old Data on GVL after a online change or change on the variable diNrOfEMS_IDOD
IF diNrOfEMS_IN <> diNrOfEMS_IN_CP AND iStateGVLData = 0 THEN iStateGVLData := 10; END_IF 

CASE iStateGVLData OF
	
	0://Init Step
		byWaitInStep := 0;
			diCounterForGVL := 1;
	
	1://Wait for 4 Steps before clean al Data on GVL
		byWaitInStep := byWaitInStep + 1;
			IF byWaitInStep >= 4 AND fbNumberDevice.bNumberIsCalculatet THEN iStateGVLData := 2; END_IF
				//To much Devices, back to the Init step
				IF byWaitInStep >= 4 AND NOT fbNumberDevice.bNumberIsCalculatet THEN iStateGVLData := 0; END_IF	
			
	2://Clear all Data in GVL
		FOR diLPForGVL := 1 TO Constants_Energy.diMaxNumberOfEMS BY 1 DO 
			Lynus_Standards.GVL_Energy.stDataGridConnections[diLPForGVL,diCounterForGVL].bEnabled := FALSE;
				Lynus_Standards.GVL_Energy.stDataGridConnections[diLPForGVL,diCounterForGVL].byErrorWarning := 0;
					Lynus_Standards.GVL_Energy.stDataGridConnections[diLPForGVL,diCounterForGVL].lrPower := 0;
						Lynus_Standards.GVL_Energy.stDataGridConnections[diLPForGVL,diCounterForGVL].lrPowerConsumption := 0;
							Lynus_Standards.GVL_Energy.stDataGridConnections[diLPForGVL,diCounterForGVL].lrPowerProduction := 0;
								Lynus_Standards.GVL_Energy.stDataGridConnections[diLPForGVL,diCounterForGVL].rSizeGridConn := 0;
		END_FOR
			diCounterForGVL := diCounterForGVL + 1;
				diCounterForGVL := LIMIT(0,diCounterForGVL,Constants_Energy.diMaxNumberOfGridConnections);
					//Back to the init step
					IF diCounterForGVL >= Constants_Energy.diMaxNumberOfGridConnections THEN iStateGVLData := 0; END_IF

	10://Clear old Data on GVL 	
		Lynus_Standards.GVL_Energy.stDataGridConnections[diNrOfEMS_IN_CP,diNrOfGrid_OUT].bEnabled := FALSE;
			Lynus_Standards.GVL_Energy.stDataGridConnections[diNrOfEMS_IN_CP,diNrOfGrid_OUT].byErrorWarning := 0;
				Lynus_Standards.GVL_Energy.stDataGridConnections[diNrOfEMS_IN_CP,diNrOfGrid_OUT].lrPower := 0;
					Lynus_Standards.GVL_Energy.stDataGridConnections[diNrOfEMS_IN_CP,diNrOfGrid_OUT].lrPowerConsumption := 0;
						Lynus_Standards.GVL_Energy.stDataGridConnections[diNrOfEMS_IN_CP,diNrOfGrid_OUT].lrPowerProduction := 0;
							Lynus_Standards.GVL_Energy.stDataGridConnections[diNrOfEMS_IN_CP,diNrOfGrid_OUT].rSizeGridConn := 0;
	
		diNrOfEMS_IN_CP := diNrOfEMS_IN;
			//Back to the init step
			iStateGVLData := 0;

END_CASE 	 

IF diNrOfGrid_OUT > 0 AND fbNumberDevice.bNumberIsCalculatet AND diNrOfEMS_IN > 0 THEN
	Lynus_Standards.GVL_Energy.stDataGridConnections[diNrOfEMS_IN,diNrOfGrid_OUT].bEnabled := fbGrid.stDataGridOut.bEnabled;
		Lynus_Standards.GVL_Energy.stDataGridConnections[diNrOfEMS_IN,diNrOfGrid_OUT].byErrorWarning := fbGrid.stDataGridOut.byErrorWarning;
			Lynus_Standards.GVL_Energy.stDataGridConnections[diNrOfEMS_IN,diNrOfGrid_OUT].lrPower := fbGrid.stDataGridOut.lrPower;
				Lynus_Standards.GVL_Energy.stDataGridConnections[diNrOfEMS_IN,diNrOfGrid_OUT].lrPowerConsumption := fbGrid.stDataGridOut.lrPowerConsumption;
					Lynus_Standards.GVL_Energy.stDataGridConnections[diNrOfEMS_IN,diNrOfGrid_OUT].lrPowerProduction := fbGrid.stDataGridOut.lrPowerProduction;
						Lynus_Standards.GVL_Energy.stDataGridConnections[diNrOfEMS_IN,diNrOfGrid_OUT].rSizeGridConn := fbGrid.stDataGridOut.rSizeGridConn;
END_IF

(*----------------------------------------------------------Save persistent data----------------------------------------------------------------*)

arrPD[1](lrValue:= BOOL_TO_LREAL(bEnable), bEventBasedActive=> );
arrPD[2](lrValue:= DINT_TO_LREAL(diNrOfEMS_IN), bEventBasedActive=> );
arrPD[3](lrValue:= DINT_TO_LREAL(diNrOfEM_IN_Grid), bEventBasedActive=> );
arrPD[4](lrValue:= REAL_TO_LREAL(rSizeGridConn), bEventBasedActive=> );
arrPD[5](lrValue:= DINT_TO_LREAL(diNrOfEMS_IN_CP), bEventBasedActive=> );

END_FUNCTION_BLOCK

// ---- FBs/Heating Pump/Linear Modular AO/FB_HP_Linear_Modular_AO.TcPOU
FUNCTION_BLOCK FB_HP_Linear_Modular_AO
VAR_INPUT PERSISTENT
	bEnable									: BOOL;												//{#lynus.ag#()} //Enable the Fuctionblock and his logic
	bPowerDataInvers						: BOOL;												//With True its possible to invert all received power data from the electric meter
	bNoLinear								: BOOL;												//Output Power from the device is not linear. Use the Values from the Table Of Interpolation Points.
	diNrOfEMS_IN							: DINT;												//Number of EMS what control this Device.
	diNrOfEM_IN_HP							: DINT;												//Number of the electric meter for incoming power data. (Power Data for this Device)
	stSetupHP								: ST_Setup_HP;										//{#lynus.ag#()} //Setup heating pump
	arrTableOfInterpolationPoints			: ARRAY[1..10] OF REAL;								//Table Of Interpolation Points. Corresponds to the different power values in the non-linear curve of the device. The last value must correspond to the maximum power.
END_VAR
VAR_INPUT
END_VAR
VAR_OUTPUT
	stDataHP								: ST_HP_Output;										//{#lynus.ag#()} //Output Data Heating pump
	diNrOfHP_OUT							: DINT;												//Active Number from the heating pump for using on other functions	
	rTargetPowerForExtFunc					: REAL;												//Target Power from 0% to +100% to use on a external Function	
END_VAR
VAR
	{attribute 'hide'}
	fbHP									: FB_HeatingPump;									//Function block for heating pump
	{attribute 'hide'}
	fbNumberDevice							: FB_NumberOfDevice;								//Function block to calcualte the number of the Device
	{attribute 'hide'}
	fbInterpolation							: FB_Lin_Interpolation;								//Function for interpolation
	fbDIExternalLock						: FB_XL1XXX_DI;										//Digital Input from external loock signal
	fbDIErrorHP								: FB_XL1XXX_DI;										//Digital Input for error from the heating pump
	{attribute 'hide'}
	timDissableFunctions					: TON;												//Timer to dissable the Function after Lynus_Standards.Constants_General.tTimeDissableLynusFunctions Days without connection to the Lynus Cloud
	{attribute 'hide'}
	timResetConnectionOnGVL					: TON;												//Timer to try reset the connection Flag on the GVL. (When somebody delete the Connection Function and make only a onlinechange)
	fbAOHP									: FB_XL4XXX_AO;										//Analog Output to swtich on and off and controll the HP
	{attribute 'hide'}
	timGetTime								: TON;												//Timer to activate the function tho read out the windows system time
	{attribute 'hide'}
	FNReset									: F_TRIG;											//Internal negative edge
	{attribute 'hide'}
	fbGetSystemTime							: NT_GetTime;										//Function to read out the windows system time on the local plc
	{attribute 'hide'}
	arrPD									: ARRAY[1..31] OF FB_PersistentData_Number;			//Function to save persistent data
	{attribute 'hide'}
	byWaitInStep							: BYTE;												//Wait in Step before start to clean data on PLC
	{attribute 'hide'}
	iStateGVLData							: INT;												//State machine to handle the data on the GVL
	{attribute 'hide'}
	diNumberOfActiveBatterys				: DINT;												//Number of active batterys
	{attribute 'hide'}
	diNumberOfBatteryInverterInEPO			: DINT;												//Number of battery inverters that work in Emergency Power operation 
	{attribute 'hide'}
	diCounterForGVL							: DINT;												//Counter to clean old data on GVL
	{attribute 'hide'}
	diLPForGVL								: DINT;												//Loop to clean old data on GVL	
	{attribute 'hide'}
	dwSumSOC								: DWORD;											//Sum of the SOC from all batterys
	{attribute 'hide'}
	lrGridPower								: LREAL;											//Grid power in kW
	{attribute 'hide'}
	lrSizeGridConnection					: LREAL;											//Size of the complete grid connection
	{attribute 'hide'}
	liLPBatteryData							: LINT;												//Loop to check some data from batterys
	{attribute 'hide'}
	liLPInEPO								: LINT;												//Loop to check if 1 or more battery inverters build a island grid	
	{attribute 'hide'}
	liLPGridData							: LINT;												//Loop to check some grid data
END_VAR
VAR PERSISTENT
	{attribute 'conditionalshow'}
	diNrOfEMS_IN_CP							: DINT;												//Number of EMS what control this Device to compare with the original
END_VAR

//Creator : Kai Ebensperger
//Company : Lynus AG
//Date : 19.05.2021
//Version : 1.0.0.0

//With this function block its possible to control a Heating pump with a analog output signal (0-10V or 4-20mA).
//This function block can control only Heating pumps with modular target power.
//With this Function block is also possible to display the electric and thermal power from the heating pump

//NOTE for diNr.....Designation => 
//_IN = Here Data come in from other Functions or go out to other functions about the GVL
//_OUT = Here Data go out to other functions about the GVL

(*------------------------------------------------------------Limits----------------------------------------------------------------------------------*)

diNrOfEMS_IN := LIMIT(0,diNrOfEMS_IN,Constants_Energy.diMaxNumberOfEMS);
	diNrOfEM_IN_HP := LIMIT(0,diNrOfEM_IN_HP,Constants_Energy.diMaxNumberOfElectricMeters);
			
(*------------------------------------------------------------------Power Data----------------------------------------------------------------------------*)

IF NOT bPowerDataInvers THEN
	fbHP.lrCounterEnergyT1_Consumption := Lynus_Standards.GVL_Energy.stDataElectricMeters[diNrOfEM_IN_HP].lrCounterEnergyT1_Production * 1000;
	fbHP.lrCounterEnergyT2_Consumption := Lynus_Standards.GVL_Energy.stDataElectricMeters[diNrOfEM_IN_HP].lrCounterEnergyT2_Production * 1000;
	fbHP.lrCounterEnergyT1_Production := Lynus_Standards.GVL_Energy.stDataElectricMeters[diNrOfEM_IN_HP].lrCounterEnergyT1_Consumption * 1000;
	fbHP.lrCounterEnergyT2_Production := Lynus_Standards.GVL_Energy.stDataElectricMeters[diNrOfEM_IN_HP].lrCounterEnergyT1_Consumption * 1000;
	fbHP.lrTotalCounterEnergy_Consumption := Lynus_Standards.GVL_Energy.stDataElectricMeters[diNrOfEM_IN_HP].lrTotalCounterEnergy_Production * 1000;
	fbHP.lrTotalCounterEnergy_Production := Lynus_Standards.GVL_Energy.stDataElectricMeters[diNrOfEM_IN_HP].lrTotalCounterEnergy_Consumption * 1000;
		fbHP.lrElPowerHP := (Lynus_Standards.GVL_Energy.stDataElectricMeters[diNrOfEM_IN_HP].lrPower * 1000) * - 1;
ELSE
	fbHP.lrCounterEnergyT1_Consumption := Lynus_Standards.GVL_Energy.stDataElectricMeters[diNrOfEM_IN_HP].lrCounterEnergyT1_Consumption * 1000;
	fbHP.lrCounterEnergyT2_Consumption := Lynus_Standards.GVL_Energy.stDataElectricMeters[diNrOfEM_IN_HP].lrCounterEnergyT2_Consumption * 1000;
	fbHP.lrCounterEnergyT1_Production := Lynus_Standards.GVL_Energy.stDataElectricMeters[diNrOfEM_IN_HP].lrCounterEnergyT1_Production * 1000;
	fbHP.lrCounterEnergyT2_Production := Lynus_Standards.GVL_Energy.stDataElectricMeters[diNrOfEM_IN_HP].lrCounterEnergyT2_Production * 1000;
	fbHP.lrTotalCounterEnergy_Consumption := Lynus_Standards.GVL_Energy.stDataElectricMeters[diNrOfEM_IN_HP].lrTotalCounterEnergy_Consumption * 1000;
	fbHP.lrTotalCounterEnergy_Production := Lynus_Standards.GVL_Energy.stDataElectricMeters[diNrOfEM_IN_HP].lrTotalCounterEnergy_Production * 1000;
		fbHP.lrElPowerHP := Lynus_Standards.GVL_Energy.stDataElectricMeters[diNrOfEM_IN_HP].lrPower * 1000;
END_IF

(*-------------------------------------------------------------Calcualte the number of HP---------------------------------------------------------------*)

fbNumberDevice(
	diActualNumberOfDevices:= Lynus_Standards.GVL_Energy.stNumberOfDevices.diNumberOfHP, 
	diMaxNumberOfDevices:= Constants_Energy.diMaxNumberOfHeatingPumps, 
	udiCounterOnlineChange:= TwinCAT_SystemInfoVarList._AppInfo.OnlineChangeCnt, 
	bNumberIsCalculatet=> , 
	bFPNumberIsCalculatet=> , 
	bOnlineChange=> , 
	diNumberForThisDevice=> diNrOfHP_OUT, 
	diNumberOfTotalDevices=> );

//Write new Numer on GVL
IF fbNumberDevice.bFPNumberIsCalculatet THEN
	Lynus_Standards.GVL_Energy.stNumberOfDevices.diNumberOfHP := fbNumberDevice.diNumberOfTotalDevices;	
END_IF 

//Delete old Number on GVL
IF fbNumberDevice.bOnlineChange THEN 
	Lynus_Standards.GVL_Energy.stNumberOfDevices.diNumberOfHP := diNrOfHP_OUT;	
		iStateGVLData := 1; 
END_IF

(*-------------------------------------------------------------Get the local windows system time for this plc---------------------------------------------------------------*)
timGetTime(IN:= bEnable AND NOT timGetTime.Q, PT:= T#30S, Q=> , ET=> );

fbGetSystemTime(
	NETID:= , 
	START:= timGetTime.Q AND NOT fbGetSystemTime.BUSY, 
	TMOUT:= , 
	BUSY=> , 
	ERR=> , 
	ERRID=> , 
	TIMESTR=> );	

fbHP.stSystemTime.wHour := fbGetSystemTime.TIMESTR.wHour;
	fbHP.stSystemTime.wMinute := fbGetSystemTime.TIMESTR.wMinute;	

(*-------------------------------------------------------------Service from Backend is ready and check the connection to backen for dissabel/enable Function---------------------------------------------------------------*)

//Try to reset the variable for connection on the GVL. When all is normal then the Lynus Mqtt connection function set this variable to true in the next cycle
//When we have no connection to the backend then after Lynus_Standards.Constants_General.tTimeDissableLynusFunctions days the Function is dissabled with all of his functionalities
timResetConnectionOnGVL(IN:= NOT timResetConnectionOnGVL.Q, PT:= T#1H, Q=> , ET=> );
	IF timResetConnectionOnGVL.Q THEN Lynus_Standards.GVL_Communicator.bStateConnectionToEnableFunctions := FALSE; END_IF
		IF NOT Lynus_Standards.GVL_Communicator.bStateConnectionToEnableFunctions THEN timDissableFunctions.IN := TRUE; ELSE timDissableFunctions.IN := FALSE; END_IF  
			timDissableFunctions(IN:= , PT:= Lynus_Standards.Constants_General.tTimeDissableLynusFunctions, Q=> , ET=> );	
	
(*------------------------------------------------------------------Error and Reset----------------------------------------------------------------------------*)	

fbDIErrorHP(bInvers:= FALSE, bSignal=> );

IF timDissableFunctions.Q THEN fbHP.bWarning := TRUE; fbHP.iWarningCode := 0; ELSE fbHP.bWarning := FALSE; END_IF 	
	IF Lynus_Standards.GVL_Energy.stNumberOfDevices.diNumberOfHP > Constants_Energy.diMaxNumberOfHeatingPumps OR fbDIErrorHP.bSignal OR fbGetSystemTime.ERR THEN fbHP.bError := TRUE; ELSE fbHP.bError := FALSE; END_IF 

IF Lynus_Standards.GVL_Energy.stNumberOfDevices.diNumberOfHP > Constants_Energy.diMaxNumberOfHeatingPumps THEN fbHP.iErrorCode := 1;
ELSIF fbGetSystemTime.ERR THEN fbHP.iErrorCode := 2; 
ELSIF fbDIErrorHP.bSignal THEN fbHP.iErrorCode := 0;
END_IF

FNReset(CLK:= fbHP.stDataHPOut.bSReset, Q=> );

(*------------------------------------------------------------------Logic----------------------------------------------------------------------------*)

//Calcualte the total SOC if we have more then 1 battery in our system
diNumberOfActiveBatterys := 0;
	dwSumSOC := 0;
		FOR liLPBatteryData := 1 TO Constants_Energy.diMaxNumberOfBatterys BY 1 DO
			IF Lynus_Standards.GVL_Energy.stDataOfBatterys[diNrOfEMS_IN,liLPBatteryData].bEnabled THEN diNumberOfActiveBatterys := diNumberOfActiveBatterys + 1; END_IF
				dwSumSOC := dwSumSOC + Lynus_Standards.GVL_Energy.stDataOfBatterys[diNrOfEMS_IN,liLPBatteryData].dwSOC;
		END_FOR
	
IF diNumberOfActiveBatterys > 0 THEN
	fbHP.dwBatterySOC := DINT_TO_DWORD(DWORD_TO_DINT(dwSumSOC) / diNumberOfActiveBatterys);
ELSE
	fbHP.dwBatterySOC := 100;	//When we have no battery in the ems system
END_IF

//Check if one or more Batterysystems or batteryinverter make island mode
diNumberOfBatteryInverterInEPO := 0;
	FOR liLPInEPO := 1 TO Constants_Energy.diMaxNumberOfBatteryInverters BY 1 DO
		IF Lynus_Standards.GVL_Energy.stDataOfBatteryInverters[diNrOfEMS_IN,liLPInEPO].bWorkOnIslandMode THEN fbHP.bEPOIsActive := TRUE; diNumberOfBatteryInverterInEPO := diNumberOfBatteryInverterInEPO + 1; END_IF
	END_FOR 
		IF diNumberOfBatteryInverterInEPO <= 0 THEN fbHP.bEPOIsActive := FALSE; END_IF

//Check the max. power of the grid connection and the sum of grid power
lrSizeGridConnection := 0;
	lrGridPower := 0;
		FOR liLPGridData := 1 TO Constants_Energy.diMaxNumberOfGridConnections BY 1 DO
			lrSizeGridConnection := lrSizeGridConnection + Lynus_Standards.GVL_Energy.stDataGridConnections[diNrOfEMS_IN,liLPGridData].rSizeGridConn;
				lrGridPower := lrGridPower + Lynus_Standards.GVL_Energy.stDataGridConnections[diNrOfEMS_IN,liLPGridData].lrPower;
		END_FOR		

//Set the target power from the EMS to the HP Function
fbHP.arrTargetPower[1] := Lynus_Standards.GVL_Energy.stDataHeatingPumps[diNrOfEMS_IN,diNrOfHP_OUT].arrTargetPowerEMS[1];

	stSetupHP.rMaxPower2 := 0;
		fbHP.arrTargetPower[2] := 0;	

//Feedback for HP is running
IF fbHP.arrTargetPower[1] > 0 THEN fbHP.bHPIsRunning := TRUE; ELSE fbHP.bHPIsRunning := FALSE; END_IF  
		
//Digital input for external lock signal
fbDIExternalLock(bInvers:= FALSE, bSignal=> );

//Functionblock HP
fbHP(
	bEnable:= bEnable AND NOT timDissableFunctions.Q, 
	bError:= , 
	bWarning:= , 
	bIsStepSwitched:= FALSE, 
	bEPOIsActive:= , 
	bExternalLock:= fbDIExternalLock.bSignal, 
	bReset:= FNReset.Q, 
	bExternalOnCommand:= Lynus_Standards.GVL_Energy.stDataHeatingPumps[diNrOfEMS_IN,diNrOfHP_OUT].bExternalOnCommand, 
	bWriteWithDelay:= TRUE, 
	bHPIsRunning:= ,
	iErrorCode:= , 
	iWarningCode:= , 
	dwBatterySOC:= , 
	diNumberOfHP:= diNrOfHP_OUT, 
	rBoilerTempHeatingSys:= 0, 
	rBoilerTempServiceWater:= 0, 
	rFlowTemp:= 0, 
	rReturnTemp:= 0, 
	rFlowTempEnergySource:= 0, 
	rReturnTempEnergySource:= 0, 
	lrSizeGridConnection:= lrSizeGridConnection, 
	lrGridPower:= lrGridPower, 
	lrTotalCounterEnergy_Consumption:= , 
	lrTotalCounterEnergy_Production:= , 
	lrCounterEnergyT1_Consumption:= , 
	lrCounterEnergyT2_Consumption:= , 
	lrCounterEnergyT1_Production:= , 
	lrCounterEnergyT2_Production:= , 
	lrCounterThermalEnergy_Heating:= 0, 
	lrCounterThermalEnergy_Water:= 0, 
	lrElPowerHP:= , 
	arrTargetPower:= , 
	tOnDelayExternalOn:= T#2M, 
	tOffDelayExternalOn:= T#2H, 
	tMinOnTime:= T#1.5H,
	tTimDelayOutput:= T#5S, 
	stSystemTime:= , 
	stSetupHP:= stSetupHP, 
	stDataHPOut=> , 
	stDataHPOutDelay=> stDataHP, 
	arrPercentValuesSteps=> );
	
(*-------------------------------------------------------------------------Output----------------------------------------------------------------------*)

IF bNoLinear THEN 
	fbInterpolation.rXInputValue := (stSetupHP.rMaxPower1 * fbHP.stDataHPOut.rTargetPower) / 100; 
		fbInterpolation.arrYIntermediateValues[1] := 10;
			fbInterpolation.arrYIntermediateValues[2] := 20;
				fbInterpolation.arrYIntermediateValues[3] := 30;
					fbInterpolation.arrYIntermediateValues[4] := 40;
						fbInterpolation.arrYIntermediateValues[5] := 50;
	fbInterpolation.arrYIntermediateValues[6] := 60;
		fbInterpolation.arrYIntermediateValues[7] := 70;
			fbInterpolation.arrYIntermediateValues[8] := 80;
				fbInterpolation.arrYIntermediateValues[9] := 90;
					fbInterpolation.arrYIntermediateValues[10] := 100;
	fbInterpolation(rXInputValue:=, arrXIntermediateValues:= arrTableOfInterpolationPoints, arrYIntermediateValues:=, rYOutputValue=> );
END_IF

IF bNoLinear THEN 
	fbAOHP.rSignal := fbInterpolation.rYOutputValue;
	//Target Power, to use this on a external Function
	rTargetPowerForExtFunc := fbInterpolation.rYOutputValue;
ELSE
	fbAOHP.rSignal := fbHP.stDataHPOut.rTargetPower;
	//Target Power, to use this on a external Function
	rTargetPowerForExtFunc := fbHP.stDataHPOut.rTargetPower;
END_IF

fbAOHP(
	rYMinTerminalValue:= 0, 
	rXMinInputSignal:= 0, 
	rYMaxTerminalValue:= 32767, 
	rXMaxInputSignal:= 100, 
	rSignal:= , 
	usiState=> );

(*-----------------------------------------------------------Handle data to Global structure for the heating pump-----------------------------------------------------------------*)

//Delte al old Data on GVL after a online change or change on the variable diNrOfEMS_IDOD
IF diNrOfEMS_IN <> diNrOfEMS_IN_CP AND iStateGVLData = 0 THEN iStateGVLData := 10; END_IF 

CASE iStateGVLData OF
	
	0://Init Step
		byWaitInStep := 0;
			diCounterForGVL := 1;
	
	1://Wait for 4 Steps before clean al Data on GVL
		byWaitInStep := byWaitInStep + 1;
			IF byWaitInStep >= 4 AND fbNumberDevice.bNumberIsCalculatet THEN iStateGVLData := 2; END_IF
				//To much Devices, back to the Init step
				IF byWaitInStep >= 4 AND NOT fbNumberDevice.bNumberIsCalculatet THEN iStateGVLData := 0; END_IF	
			
	2://Clear all Data in GVL
		FOR diLPForGVL := 1 TO Constants_Energy.diMaxNumberOfEMS BY 1 DO
			Lynus_Standards.GVL_Energy.stDataHeatingPumps[diLPForGVL,diCounterForGVL].bEnabled := FALSE;
				Lynus_Standards.GVL_Energy.stDataHeatingPumps[diLPForGVL,diCounterForGVL].arrMaxPower[1] := 0;
					Lynus_Standards.GVL_Energy.stDataHeatingPumps[diLPForGVL,diCounterForGVL].arrMaxPower[2] := 0;
						Lynus_Standards.GVL_Energy.stDataHeatingPumps[diLPForGVL,diCounterForGVL].bIsControllable := FALSE;
							Lynus_Standards.GVL_Energy.stDataHeatingPumps[diLPForGVL,diCounterForGVL].bIsStepSwitched := FALSE;
								Lynus_Standards.GVL_Energy.stDataHeatingPumps[diLPForGVL,diCounterForGVL].byErrorWarning := 0;
									Lynus_Standards.GVL_Energy.stDataHeatingPumps[diLPForGVL,diCounterForGVL].byNumberOfSteps := 0;
										Lynus_Standards.GVL_Energy.stDataHeatingPumps[diLPForGVL,diCounterForGVL].byPriority := 0;
											Lynus_Standards.GVL_Energy.stDataHeatingPumps[diLPForGVL,diCounterForGVL].lrElPower := 0;
												Lynus_Standards.GVL_Energy.stDataHeatingPumps[diLPForGVL,diCounterForGVL].lrElPowerConsumption := 0;
													Lynus_Standards.GVL_Energy.stDataHeatingPumps[diLPForGVL,diCounterForGVL].lrElPowerProduction := 0;
														Lynus_Standards.GVL_Energy.stDataHeatingPumps[diLPForGVL,diCounterForGVL].rBoilerTempHeatingSys := 0;
															Lynus_Standards.GVL_Energy.stDataHeatingPumps[diLPForGVL,diCounterForGVL].rBoilerTempServiceWater := 0;
																Lynus_Standards.GVL_Energy.stDataHeatingPumps[diLPForGVL,diCounterForGVL].rFlowTemp := 0;
																	Lynus_Standards.GVL_Energy.stDataHeatingPumps[diLPForGVL,diCounterForGVL].rFlowTempEnergySource := 0;
																		Lynus_Standards.GVL_Energy.stDataHeatingPumps[diLPForGVL,diCounterForGVL].rReturnTemp := 0;
																			Lynus_Standards.GVL_Energy.stDataHeatingPumps[diLPForGVL,diCounterForGVL].rReturnTempEnergySource := 0;
																				//Set also the target value from ems back here to 0 and not in EMS function because EMS is in Standy when we have a online change (Problem when we delete a ems function and make a online change)
																				Lynus_Standards.GVL_Energy.stDataHeatingPumps[diLPForGVL,diCounterForGVL].arrTargetPowerEMS[1] := 0;
																					Lynus_Standards.GVL_Energy.stDataHeatingPumps[diLPForGVL,diCounterForGVL].arrTargetPowerEMS[2] := 0;
																						Lynus_Standards.GVL_Energy.stDataHeatingPumps[diLPForGVL,diCounterForGVL].bExternalOnCommand := FALSE;	
		END_FOR
			diCounterForGVL := diCounterForGVL + 1;
				diCounterForGVL := LIMIT(0,diCounterForGVL,Constants_Energy.diMaxNumberOfHeatingPumps);
					//Back to the init step
					IF diCounterForGVL >= Constants_Energy.diMaxNumberOfHeatingPumps THEN iStateGVLData := 0; END_IF

